ELSE
	tower_lamp.iol_slave_pdo_output.seg_1_color := 0; 
	tower_lamp.iol_slave_pdo_output.seg_2_color := 0; 
	tower_lamp.iol_slave_pdo_output.seg_3_color := 0; 
	
END_IF
*)
(*************************************************************************************
**************************************************************************************)

_handle_messages();
_write_output();

ACTION _handle_messages:
;
END_ACTION

ACTION _handle_process_test:
;
END_ACTION

ACTION _mode_manager:
IF process_mode_req_is_pending(CONVERSION_this := prc)
THEN
    process_apply_mode_req_first_step(CONVERSION_this := prc);
    CASE process_get_mode(CONVERSION_this := prc) OF
        MODE_TO_ABSENT:
            ;
        MODE_TO_INACTIVE:
            ;
        MODE_TO_TEST:
            ;
        MODE_TO_OPERATIONAL:
            ;
    END_CASE
    process_apply_mode_req_second_step(CONVERSION_this := prc);
END_IF;
END_ACTION

ACTION _objects_manager:
IF objects_initialization()
THEN
    sub_process_init(
        object_name 				:= 'csp_main_services_towerLamp.prc',
        process						:= csp_main_services.prc,
        CONVERSION_this				:= prc);

	prc_path 						:= process_get_path(prc);

	digital_output_init(
		object_name 				:= CONCAT(prc_path, '_buzzer_do'),
		polarity_direct				:= TRUE,
		process 					:= prc,
		CONVERSION_this 			:= buzzer_do);
		
	lamp_init(
		object_name 				:= CONCAT(prc_path, '_buzzer_lmp'),
		process 					:= prc,
		dout						:= buzzer_do,
		CONVERSION_this 			:= buzzer_lmp);
	
	filter_init(
		object_name := CONCAT(prc_path, '_buzzer_filt'),
		delay_off_on := 0,
		delay_on_off := 3000, //Marco: it's equal to the half of the desired buzzer timer (i.e. desired 1.5s --> delay = 3 s)
		process := prc,
		CONVERSION_this := buzzer_filt);
	
		(* BUZZER CONDITIONER *)
	motorization_conditioner_init(
		object_name					:= CONCAT(prc_path, '_buzzer_motcond'),
		velocity_limit				:= 0.0,
		velocity_limit_active		:= FALSE,
		idle_handshake_active		:= FALSE,
		execute_handshake_active	:= TRUE,
		hold_handshake_active		:= FALSE,
		suspend_handshake_active	:= FALSE,
		complete_handshake_active	:= FALSE,
		abort_handshake_active		:= FALSE,
		stop_handshake_active		:= FALSE,
		origin						:= MOTORIZATION_CONDITIONER_ORIGIN_INTERNAL,
		manager						:= csp_main_motorization_manager.motm,
		process						:= prc,
		CONVERSION_this				:= buzzer_motcond);

	boolean_or_init(
		object_name 				:= CONCAT(prc_path, '_buzzer_req_bool_or'),
		process 					:= prc,
		CONVERSION_this 			:= buzzer_req_bool_or);
	
	(* boolean_init(            
		object_name					:= CONCAT(prc_path, '_buzzer_status_bool'), 
		process						:= prc, 
		CONVERSION_this				:= buzzer_status_bool);
		
	signaling_device_configure_buzzer_behaviour(
		working_mode:= SIGNALING_DEVICE_BUZZER_WORKING_MODE_STATE_ON_OFF, 
		custom_pwm_period_ms:= 0, 
		buzzer_time_to_exec_from_starting:=3000 , 
		buzzer_time_to_exec_from_unholding:= 300, 
		CONVERSION_this:=tower_lamp );

	timer_init(
		object_name					:= CONCAT(prc_path, '_buzzer_tmr'),
		process						:= prc,
	    CONVERSION_this				:= buzzer_tmr);


		*)	
		
	signaling_device_iol_balluff_init(
		object_name 				:= CONCAT(prc_path, '_tower_lamp'),
		master_channel 				:= 1,
		blue_light_enable 			:= TRUE,
		white_light_enable 			:= TRUE,
		io_link_master 				:= csp_main_services.iol_master_el6224_IO6100,
		machine 					:= csp.mch,
		buzzer 						:= buzzer_lmp,
		process 					:= prc,
		CONVERSION_this 			:= tower_lamp);
	
	filter_init(
		object_name 				:= CONCAT(prc_path, '_reject_status_flt'),
		delay_off_on				:= flt_timer_off_on,
		delay_on_off 				:= flt_timer_on_off,
		process			 			:= prc,
		CONVERSION_this 			:= reject_status_flt);	
	
	parameter_overwrite_bool_init(
		object_name								:= CONCAT(prc_path, '_reject_ack_overwrite'),
		parameter								:= Reject_Acknowledged,
		process									:= prc,
		CONVERSION_this							:= reject_ack_overwrite);
	
	
END_IF;

IF	objects_running()
THEN
	process_cycle(prc);
	lamp_cycle(buzzer_lmp);
	
	filter_cycle(input:= buzzer_req_bool, buzzer_filt);
	filter_cycle(input:= reject_present_filtered,	CONVERSION_this := reject_status_flt);	
		
	signaling_device_cycle(tower_lamp);
	motorization_conditioner_cycle(buzzer_motcond);
END_IF;
END_ACTION

ACTION _read_process_image:
;
END_ACTION

ACTION _read_var_input:
;
END_ACTION

ACTION _set_runtime_properties:
;
END_ACTION

ACTION _sim_update:
;
END_ACTION

ACTION _write_output:
(* SIMULATION *)
;
END_ACTION

END_PROGRAM

// ---- Application/CSP/Main/Services/csp_main_services.TcPOU
(********************* G.D S.p.A. - Technical Department *****************************

Date			Version		Author			Description             
----------      -------		-----------		----------------------------------------------
2015/06/30		0000.00		M.Grasso		Initial Release

DESCRIPTION:	

NOTES:        		 

**************************************************************************************)
(*$R process_ref := prc; $*)

PROGRAM csp_main_services
VAR
	prc:								process;
	prc_path:							STRING;
	reset_output_test:					digital_output;
	
	iol_master_el6224_IO6100:			iol_master;
	
	lights_toggle:						BOOL := TRUE; (*$P $*)
	
	pressure_switch_value AT %I*:		INT;
	no_pressure_dchk:					digital_check;
	pressure_level_low_bool:			boolean;
	pressure_value_limit:				INT := 1000; (*$P $*)
	pressure_check_delay:				DINT := 15000; (*$P $*)
	
	air_not_above_limit_motcond:		motorization_conditioner;
	
	pressure_check_delay_running: 		DINT := 100;
END_VAR

_read_var_input();
_objects_manager();

IF g_application_status <> APPLICATION_STATUS_RUNNING
THEN
	RETURN;
END_IF

_read_process_image();

_mode_manager();

CASE process_get_mode (CONVERSION_this := prc) OF

	MODE_ABSENT,
	MODE_INACTIVE:
		RETURN;

	MODE_TEST:
		_handle_process_test();
END_CASE
_set_runtime_properties();

(*************************************************************************************
**************************************************************************************)
(*BODY*)

IF descriptor_get_reset_edge(prc.descriptor)
THEN
	digital_output_set(reset_output_test);
ELSE
	digital_output_reset(reset_output_test);
END_IF



(* LOGIC TO CHECK FOR PRESSURE AFTER MACHINE IS READY *)
IF machine_is_running(csp.mch)
AND pressure_switch_value < pressure_value_limit
	THEN
		digital_check_set_alarm_delay(
			alarm_delay := pressure_check_delay_running,
			CONVERSION_this := no_pressure_dchk);
		boolean_set(pressure_level_low_bool);
END_IF

IF machine_is_ready(csp.mch)
AND pressure_switch_value < pressure_value_limit
	THEN
digital_check_set_alarm_delay(
	alarm_delay := pressure_check_delay,
	CONVERSION_this := no_pressure_dchk);
		boolean_set(pressure_level_low_bool);
END_IF


IF machine_is_stopped(csp.mch)
	OR 
	pressure_switch_value > pressure_value_limit
	THEN
	boolean_reset(pressure_level_low_bool);
END_IF



IF	motorization_manager_is_starting(csp_main_motorization_manager.motm)
AND pressure_switch_value > pressure_value_limit
	THEN
		motorization_conditioner_start_done(air_not_above_limit_motcond);
END_IF

(*************************************************************************************
**************************************************************************************)

_handle_messages();
_write_output();

ACTION _handle_messages:
;
END_ACTION

ACTION _handle_process_test:
;
END_ACTION

ACTION _mode_manager:
IF process_mode_req_is_pending(CONVERSION_this := prc)
THEN
    process_apply_mode_req_first_step(CONVERSION_this := prc);
    CASE process_get_mode(CONVERSION_this := prc) OF
        MODE_TO_ABSENT:
            ;
        MODE_TO_INACTIVE:
            ;
        MODE_TO_TEST:
            ;
        MODE_TO_OPERATIONAL:
            ;
    END_CASE
    process_apply_mode_req_second_step(CONVERSION_this := prc);
END_IF;
END_ACTION

ACTION _objects_manager:
IF objects_initialization()
THEN
    sub_process_init(
	    object_name 	:= 'csp_main_services.prc',
        process			:= csp_main.prc,
        CONVERSION_this			:= prc);

	prc_path 			:= process_get_path(prc);

	digital_output_init(
		object_name		:= CONCAT(prc_path, '_reset_output_test'),
		polarity_direct	:= TRUE,
		process			:= prc,
		CONVERSION_this	:= reset_output_test);
		
	iol_master_init(
		object_name := 			'iol_master_el6224_IO6100',
		device_name := 			'SPLC5000Slot19 (EL6224)',
		_type := 				IOL_MASTER_BECKHOFF_EL6224,
		ethercat_master :=		csp_main.cabinet_ethercat_master,
		process := 				prc,
		CONVERSION_this := 		iol_master_el6224_IO6100);
		
		
	digital_check_and_message_init(
		object_name			:= CONCAT(prc_path, '_no_pressure_dchk'),
		alarm_if_input_off	:= FALSE,
		alarm_delay			:= pressure_check_delay,
		enabled_at_powerup	:= TRUE,
		individual_reset	:= FALSE,
		machine_reaction	:= MACHINE_REACTION_EMERGENCY_STOP,
		typology			:= MESSAGE_TYPOLOGY_EMERGENCY,
		process				:= prc,
		CONVERSION_this		:= no_pressure_dchk);

	boolean_init(
		object_name			:= CONCAT(prc_path, '_pressure_level_boolean'),
		process				:= prc,
		CONVERSION_this		:= pressure_level_low_bool);

	digital_check_add_boolean(
		boolean				:= pressure_level_low_bool,
		CONVERSION_this		:= no_pressure_dchk);

		
	motorization_conditioner_init(
		object_name					:=	CONCAT(prc_path, '_air_not_above_limit_motcond'),
		velocity_limit				:=	0.0,
		velocity_limit_active		:=	FALSE,
		idle_handshake_active		:=	FALSE,
		execute_handshake_active	:=	TRUE,
		hold_handshake_active		:=	FALSE,
		suspend_handshake_active	:=	FALSE,
		complete_handshake_active	:=	FALSE,
		abort_handshake_active		:=	FALSE,
		stop_handshake_active		:=	FALSE,
		origin						:=	MOTORIZATION_CONDITIONER_ORIGIN_INTERNAL,
		manager						:=	csp_main_motorization_manager.motm,
		process						:=	prc,
		CONVERSION_this				:=	air_not_above_limit_motcond);
		
END_IF

IF objects_running()
THEN
	process_cycle(prc);
	iol_master_cycle(iol_master_el6224_IO6100);
	digital_check_cycle(no_pressure_dchk);
	motorization_conditioner_cycle(air_not_above_limit_motcond);
END_IF
END_ACTION

ACTION _read_process_image:
;
END_ACTION

ACTION _read_var_input:
;
END_ACTION

ACTION _set_runtime_properties:
;
END_ACTION

ACTION _write_output:
;
END_ACTION

END_PROGRAM

// ---- Application/CSP/Case/Feed/Kinematic/csp_case_feed_kinematic_y.TcPOU
(*********************************** G.D S.p.A. - Technical Department ***********************************
============= PROGRAM INFO ============
FOLDER:             TBD
MACHINES INVOLVED:  TBD 

============= DESCRIPTION =============
csp machine declaration

============= REVISIONS ===============
Date		Version	 	Author      	Description             
----------	-------		------------  	--------------------------------------------
2019/04/05 	0000.00	 	M.Grasso		Creation of the PRG

**********************************************************************************************************)
(*$R process_ref := prc; $*)
PROGRAM csp_case_feed_kinematic_y
VAR
		
	prc:												process;
	prc_path:											STRING;
	
	axis:												axis;
	axis_actual_position:								LREAL;

	fsm_enable_condition:								BOOL := FALSE;
	fsm_next_status:									csp_case_feed_kinematic_status_enum;
	fsm_status:											csp_case_feed_kinematic_status_enum;
	debug_state_machine:								BOOL := FALSE;
	debug_state_machine_one_step:						BOOL := FALSE;	
	
	in_accu_safe_pos:                                   BOOL := FALSE;
    accu_tolerance:                                     LREAL := 5.0;
    accu_safe_pos:                                      LREAL := -485;
	
	cam_id:												INT := 3;
	
	local_test: BOOL := false;
END_VAR

VAR CONSTANT
	MOTOR_PHASE_VELOCITY_MMPS:							LREAL := 20;	
	MOTOR_MAX_VELOCITY_MMPS:							LREAL := 1000;
	MOTOR_MAX_ACCELLERATION_MMPS2:						LREAL := 10000;
	MOTOR_MAX_DECELLERATION_MMPS2:						LREAL := 10000;
	MOTOR_MAX_JERK_MMPS3:								LREAL := 100000; 
	MOTOR_MAX_FOLLOWING_ERROR_MM:						LREAL := 10;
END_VAR

_read_var_input();

_object_manager();

IF NOT objects_running()
THEN
	RETURN;	
END_IF

_read_process_image();

_mode_manager();

CASE process_get_mode(prc) OF
	MODE_ABSENT,
	MODE_INACTIVE:
		RETURN;
	MODE_TEST:
		_handle_process_test();
END_CASE

_set_runtime_properties();

(********************************* BODY *********************************)

IF (axis.actual_position > (accu_safe_pos - accu_tolerance)) AND axis.actual_position < (accu_safe_pos + accu_tolerance)
THEN
	in_accu_safe_pos := TRUE;
ELSE
	in_accu_safe_pos := FALSE;   
END_IF

// Manage the accu change safe position
fsm_enable_condition := axis_is_ok(FALSE, axis)	
						AND															
						(csp_case_feed_kinematic.fsm_status = CSP_CASE_FEED_KINEMATIC_STATUS_ENABLED)
						AND
						csp_case_feed_kinematic.cartesian_mode_active
						AND							
						csp_main_accuChange.Brand_Change_Occurred;
										
IF	NOT fsm_enable_condition
	AND
	fsm_status <> CSP_CASE_FEED_KINEMATIC_STATUS_DISABLED	
THEN
	fsm_next_status	:= CSP_CASE_FEED_KINEMATIC_STATUS_DISABLED;
END_IF
					
CASE fsm_status OF
	
	CSP_CASE_FEED_KINEMATIC_STATUS_NOT_INITIALIZED:
	
        IF	axis_is_ok(return_when_absent := TRUE, CONVERSION_this := axis)
        THEN
            fsm_next_status := CSP_CASE_FEED_KINEMATIC_STATUS_DISABLED;
        END_IF

		
	CSP_CASE_FEED_KINEMATIC_STATUS_DISABLED:
	
		IF	fsm_enable_condition
			AND
			motorization_conditioner_is_execute(csp_main_services_towerLamp.buzzer_motcond) 							
		THEN	
			IF	in_accu_safe_pos
			THEN
				fsm_next_status := CSP_CASE_FEED_KINEMATIC_STATUS_CHANGE_OVER_MODE_DONE;
			ELSE								
				fsm_next_status := CSP_CASE_FEED_KINEMATIC_STATUS_ENABLED;
			END_IF
		END_IF;

		
	CSP_CASE_FEED_KINEMATIC_STATUS_ENABLED:	
	
		axis_move_absolute(
			position 		:= accu_safe_pos,
			velocity 		:= MOTOR_PHASE_VELOCITY_MMPS,
			direction		:= AXIS_CURRENT_DIRECTION,
			acceleration 	:= MOTOR_MAX_ACCELLERATION_MMPS2,
			deceleration 	:= MOTOR_MAX_DECELLERATION_MMPS2,
			jerk 			:= MOTOR_MAX_JERK_MMPS3, 
			buffer_mode 	:= AXIS_BUFFER_MODE_BUFFERED,
			CONVERSION_this := axis);
			
		IF 	axis_is_absolute_moving(axis)
		THEN
			fsm_next_status	:= CSP_CASE_FEED_KINEMATIC_STATUS_CHANGE_OVER_MODE;
		END_IF
		
		
	CSP_CASE_FEED_KINEMATIC_STATUS_CHANGE_OVER_MODE:

		IF 	axis_is_standstill(axis)
		THEN	
			axis_disable(axis);					
			fsm_next_status := CSP_CASE_FEED_KINEMATIC_STATUS_CHANGE_OVER_MODE_DONE;
		END_IF
		
		
	CSP_CASE_FEED_KINEMATIC_STATUS_CHANGE_OVER_MODE_DONE:
		;
		
END_CASE

IF 	NOT debug_state_machine
	OR
	debug_state_machine_one_step
THEN
	fsm_status := fsm_next_status;
	debug_state_machine_one_step := FALSE;
END_IF

(* TEMPORARY CAM CHANGE *)
IF csp_main_brand.count = '24Count'
	THEN
		cam_id := 503; //beta 1,3,10 = 303; beta 4 = 503; alpha 1 = 403
ELSIF csp_main_brand.count = '10Count'
	THEN
		cam_id := 572;
ELSIF csp_main_brand.count = '32Count'
	THEN
		cam_id := 3;
ELSIF csp_main_brand.count = '48Count'
	THEN
		cam_id := 44;
END_IF

(************************************************************************)

_handle_messages();

_write_output();

ACTION _handle_messages:
;
END_ACTION

ACTION _handle_process_test:
;
END_ACTION

ACTION _mode_manager:
IF process_mode_req_is_pending(prc)
THEN
    process_apply_mode_req_first_step(prc);
    CASE process_get_mode(prc) OF
        MODE_TO_ABSENT:
			;
        MODE_TO_INACTIVE:
			;
        MODE_TO_TEST:
			;
        MODE_TO_OPERATIONAL:
			;
    END_CASE
    process_apply_mode_req_second_step(prc);
END_IF
END_ACTION

ACTION _object_manager:
IF objects_initialization()
THEN
	sub_process_init(
		object_name					:= 'csp_case_feed_kinematic_y.prc', 
		process						:= csp_case_feed_kinematic.prc, 
		CONVERSION_this				:= prc);
		
	prc_path 						:= process_get_path(prc);
	
	axis_init(
		object_name					:= CONCAT(prc_path, '_axis'), 
		axis_type					:= AXIS_TYPE_VIRTUAL, 
		encoder_scaling_factor		:= G_VIRTUAL_ENCODER_SCALING_FACTOR_DEGPINC,
		modulo						:= G_NO_MODULO_DEG, 
		process						:= prc, 
		CONVERSION_this				:= axis);
	
	axis_set_max_dynamic(
		reference_velocity			:=	MOTOR_MAX_VELOCITY_MMPS,
		velocity					:=	MOTOR_MAX_VELOCITY_MMPS,
		acceleration				:=	MOTOR_MAX_ACCELLERATION_MMPS2,
		deceleration				:=	MOTOR_MAX_DECELLERATION_MMPS2,
		jerk						:=	MOTOR_MAX_JERK_MMPS3,
		following_error				:=	MOTOR_MAX_FOLLOWING_ERROR_MM,
		CONVERSION_this				:=	axis);
		

END_IF

IF objects_running()
THEN
	process_cycle(prc);
	axis_cycle(axis);
END_IF
END_ACTION

ACTION _read_process_image:
;
END_ACTION

ACTION _read_var_input:
;
END_ACTION

ACTION _set_runtime_properties:
axis_actual_position := axis_get_actual_incremental_position(axis);
END_ACTION

ACTION _write_output:
;
END_ACTION

END_PROGRAM

// ---- Application/CSP/Case/Feed/Kinematic/csp_case_feed_kinematic_tilt.TcPOU
(*********************************** G.D S.p.A. - Technical Department ***********************************
============= PROGRAM INFO ============
FOLDER:             TBD
MACHINES INVOLVED:  TBD 

============= DESCRIPTION =============
csp machine declaration

============= REVISIONS ===============
Date		Version	 	Author      	Description             
----------	-------		------------  	--------------------------------------------
2019/04/05 	0000.00	 	M.Grasso		Creation of the PRG

**********************************************************************************************************)
(*$R process_ref := prc; $*)
PROGRAM csp_case_feed_kinematic_tilt
VAR
		
	prc:												process;
	prc_path:											STRING;
	
	axis:												axis;
	axis_actual_position:								LREAL;
	
	fsm_enable_condition:								BOOL := FALSE;
	fsm_next_status:									csp_case_feed_kinematic_status_enum;
	fsm_status:											csp_case_feed_kinematic_status_enum;
	debug_state_machine:								BOOL := FALSE;
	debug_state_machine_one_step:						BOOL := FALSE;	
	
	in_accu_safe_pos:                                   BOOL := FALSE;
    accu_tolerance:                                     LREAL := 5.0;
    accu_safe_pos:                                      LREAL := 1334.5;
	
	cam_id:												INT := 7;

	local_test: 										BOOL := false;
END_VAR

VAR CONSTANT
	MOTOR_PHASE_VELOCITY_DEGPS:							LREAL := 8;	
	MOTOR_MAX_VELOCITY_DEGPS:							LREAL := 9600;
	MOTOR_MAX_ACCELLERATION_DEGPS2:						LREAL := 4800;
	MOTOR_MAX_DECELLERATION_DEGPS2:						LREAL := 4800;
	MOTOR_MAX_JERK_DEGPS3:								LREAL := 100000000; 
	MOTOR_MAX_FOLLOWING_ERROR_DEG:						LREAL := 2;
END_VAR

_read_var_input();

_object_manager();

IF 	NOT objects_running()
THEN
	RETURN;	
END_IF

_read_process_image();

_mode_manager();

CASE process_get_mode(prc) OF
	MODE_ABSENT,
	MODE_INACTIVE:
		RETURN;
	MODE_TEST:
		_handle_process_test();
END_CASE

_set_runtime_properties();

(********************************* BODY *********************************)

IF (axis.actual_position > (accu_safe_pos - accu_tolerance)) AND axis.actual_position < (accu_safe_pos + accu_tolerance)
THEN
	in_accu_safe_pos := TRUE;
ELSE
	in_accu_safe_pos := FALSE;   
END_IF

// Manage the accu change safe position
fsm_enable_condition := axis_is_ok(FALSE, axis)	
						AND															
						(csp_case_feed_kinematic.fsm_status = CSP_CASE_FEED_KINEMATIC_STATUS_ENABLED)
						AND
						csp_case_feed_kinematic.cartesian_mode_active
						AND							
						csp_main_accuChange.Brand_Change_Occurred;
										
IF	NOT fsm_enable_condition
	AND
	fsm_status <> CSP_CASE_FEED_KINEMATIC_STATUS_DISABLED	
THEN
	fsm_next_status	:= CSP_CASE_FEED_KINEMATIC_STATUS_DISABLED;
END_IF
					
CASE fsm_status OF
	
	CSP_CASE_FEED_KINEMATIC_STATUS_NOT_INITIALIZED:
	
        IF	axis_is_ok(return_when_absent := TRUE, CONVERSION_this := axis)
        THEN
            fsm_next_status := CSP_CASE_FEED_KINEMATIC_STATUS_DISABLED;
        END_IF
		

	CSP_CASE_FEED_KINEMATIC_STATUS_DISABLED:
	
		IF	fsm_enable_condition
			AND
			motorization_conditioner_is_execute(csp_main_services_towerLamp.buzzer_motcond) 							
		THEN	
			IF	in_accu_safe_pos
			THEN
				fsm_next_status := CSP_CASE_FEED_KINEMATIC_STATUS_CHANGE_OVER_MODE_DONE;
			ELSE								
				fsm_next_status := CSP_CASE_FEED_KINEMATIC_STATUS_ENABLED;
			END_IF
		END_IF;
		

	CSP_CASE_FEED_KINEMATIC_STATUS_ENABLED:	
	
		axis_move_absolute(
			position 		:= accu_safe_pos,
			velocity 		:= MOTOR_PHASE_VELOCITY_DEGPS,
			direction		:= AXIS_CURRENT_DIRECTION,
			acceleration 	:= MOTOR_MAX_ACCELLERATION_DEGPS2,
			deceleration 	:= MOTOR_MAX_DECELLERATION_DEGPS2,
			jerk 			:= MOTOR_MAX_JERK_DEGPS3, 
			buffer_mode 	:= AXIS_BUFFER_MODE_BUFFERED,
			CONVERSION_this := axis);
			
		IF 	axis_is_absolute_moving(axis)
		THEN
			fsm_next_status	:= CSP_CASE_FEED_KINEMATIC_STATUS_CHANGE_OVER_MODE;
		END_IF
		
		
	CSP_CASE_FEED_KINEMATIC_STATUS_CHANGE_OVER_MODE:
	
		IF 	axis_is_standstill(axis)
		THEN	
			axis_disable(axis);					
			fsm_next_status := CSP_CASE_FEED_KINEMATIC_STATUS_CHANGE_OVER_MODE_DONE;
		END_IF
		
	CSP_CASE_FEED_KINEMATIC_STATUS_CHANGE_OVER_MODE_DONE:
	
		;
		
END_CASE

IF 	NOT debug_state_machine
	OR
	debug_state_machine_one_step
THEN
	fsm_status := fsm_next_status;
	debug_state_machine_one_step := FALSE;
END_IF


(* TEMPORARY CAM CHANGE *)
IF csp_main_brand.count = '24Count'
	THEN
		cam_id := 307;
ELSIF csp_main_brand.count = '10Count'
	THEN
		cam_id := 573;
ELSIF csp_main_brand.count = '32Count'
	THEN
		cam_id := 7;
ELSIF csp_main_brand.count = '48Count'
	THEN
		cam_id := 45;
END_IF

(************************************************************************)

_handle_messages();

_write_output();

ACTION _handle_messages:
;
END_ACTION

ACTION _handle_process_test:
;
END_ACTION

ACTION _mode_manager:
IF process_mode_req_is_pending(prc)
THEN
    process_apply_mode_req_first_step(prc);
    CASE process_get_mode(prc) OF
        MODE_TO_ABSENT:
			;
        MODE_TO_INACTIVE:
			;
        MODE_TO_TEST:
			;
        MODE_TO_OPERATIONAL:
			;
    END_CASE
    process_apply_mode_req_second_step(prc);
END_IF
END_ACTION

ACTION _object_manager:
IF objects_initialization()
THEN
	sub_process_init(
		object_name					:= 'csp_case_feed_kinematic_tilt.prc', 
		process						:= csp_case_feed_kinematic.prc, 
		CONVERSION_this				:= prc);
		
	prc_path 						:= process_get_path(prc);
	
	axis_init(
		object_name					:= CONCAT(prc_path, '_axis'), 
		axis_type					:= AXIS_TYPE_VIRTUAL, 
		encoder_scaling_factor		:= G_VIRTUAL_ENCODER_SCALING_FACTOR_DEGPINC,
		modulo						:= G_NO_MODULO_DEG, 
		process						:= prc, 
		CONVERSION_this				:= axis);
	
	axis_set_max_dynamic(
		reference_velocity			:=	MOTOR_MAX_VELOCITY_DEGPS,
		velocity					:=	MOTOR_MAX_VELOCITY_DEGPS,
		acceleration				:=	MOTOR_MAX_ACCELLERATION_DEGPS2,
		deceleration				:=	MOTOR_MAX_DECELLERATION_DEGPS2,
		jerk						:=	MOTOR_MAX_JERK_DEGPS3,
		following_error				:=	MOTOR_MAX_FOLLOWING_ERROR_DEG,
		CONVERSION_this				:=	axis);
	

END_IF

IF objects_running()
THEN
	process_cycle(prc);
	axis_cycle(axis);
END_IF
END_ACTION

ACTION _read_process_image:
;
END_ACTION

ACTION _read_var_input:
;
END_ACTION

ACTION _set_runtime_properties:
axis_actual_position := axis_get_actual_incremental_position(axis);
END_ACTION

ACTION _write_output:
;
END_ACTION

END_PROGRAM

// ---- POUs/AFL extensions/jog_manager/commands/jog_manager_reset_pendant_active.TcPOU
(*$
	Reset the pendant activation to ogject <b><i>this</i></b>.
	The method returns <i>TRUE</i> if the command is accepted, otherwise it returns <i>FALSE</i>.
$*)
FUNCTION jog_manager_reset_pendant_active : BOOL
VAR_INPUT	
END_VAR
VAR_IN_OUT
    CONVERSION_this:		jog_manager;	(*$ Instance to which the method applies $*)
END_VAR

IF	NOT (descriptor_mode_is_operational(CONVERSION_this.descriptor)
		(*OR
		descriptor_mode_is_test(CONVERSION_this.descriptor)*))
THEN
	jog_manager_reset_pendant_active := FALSE;				(* command rejected *)
 	RETURN;
END_IF

parameter_overwrite_set_bool_value(FALSE, CONVERSION_this.pendant_active_pow);

jog_manager_reset_pendant_active := TRUE;					(* command accepted *)

END_FUNCTION

// ---- POUs/AFL extensions/jog_manager/status/jog_manager_is_pendant_active.TcPOU
(*$
	Returns <i>pendant_active</i> of the instance <b><i>this</i></b>.
	Returns always false if pendant is not present.
$*)
FUNCTION jog_manager_is_pendant_active: BOOL
VAR_IN_OUT
    CONVERSION_this:	jog_manager;	(*$ Instance to which the method applies $*)
END_VAR

jog_manager_is_pendant_active := 
	CONVERSION_this.has_pendant
	AND
	CONVERSION_this.pendant_active;

END_FUNCTION

// ---- Application/CSP/Case/Feed/csp_case_feed.TcPOU
(*********************************** G.D S.p.A. - Technical Department ***********************************
============= PROGRAM INFO ============
FOLDER:             TBD
MACHINES INVOLVED:  TBD 

============= DESCRIPTION =============
csp machine declaration

============= REVISIONS ===============
Date		Version	 	Author      	Description             
----------	-------		------------  	--------------------------------------------
2019/04/05 	0000.00	 	M.Grasso		Creation of the PRG

**********************************************************************************************************)
(*$R process_ref := prc; $*)
PROGRAM csp_case_feed
VAR
	
	prc:											process;
	prc_path:										STRING;
	
	Feed_request:									BOOL;
	case_at_loading_sr: 							DINT := 26;
END_VAR

_read_var_input();

_object_manager();

IF NOT objects_running()
THEN
	RETURN;	
END_IF

_read_process_image();

_mode_manager();

_set_runtime_properties();

(********************************* BODY *********************************)
IF (shift_register_step_has_status_item(
	step_id := case_at_loading_sr,
	status_bits_to_be_true := ITEM_HAS_LS_LOWER_FLAP + ITEM_HAS_LS_UPPER_FLAP + ITEM_HAS_OS_LOWER_FLAP + ITEM_HAS_OS_UPPER_FLAP,
	status_bits_to_be_false := 0,
	CONVERSION_this :=csp_case_main_statistics.sr)
   
	AND
	(csp_case_feed_virtualMaster.axis.actual_modulo_position > 340 
	AND NOT csp_case_loader_virtualMaster.product_loaded))   
	AND csp_case_loader.load_ready_at_loader	           
	THEN		 
		Feed_request :=FALSE;
	ELSIF NOT csp_case_transport_virtualMaster.stop_for_reject 
		THEN  
		Feed_request :=TRUE;
              
END_IF
(************************************************************************)

_handle_messages();

_write_output();

ACTION _handle_messages:
;
END_ACTION

ACTION _handle_process_test:
;
END_ACTION

ACTION _mode_manager:
IF process_mode_req_is_pending(prc)
THEN
    process_apply_mode_req_first_step(prc);
    CASE process_get_mode(prc) OF
        MODE_TO_ABSENT:
			;
        MODE_TO_INACTIVE:
			;
        MODE_TO_TEST:
			;
        MODE_TO_OPERATIONAL:
			;
    END_CASE
    process_apply_mode_req_second_step(prc);
END_IF
END_ACTION

ACTION _object_manager:
IF objects_initialization()
THEN
	sub_process_init(
		object_name					:= 'csp_case_feed.prc', 
		process						:= csp_case.prc, 
		CONVERSION_this				:= prc);
		
	prc_path 						:= process_get_path(prc);
END_IF

IF objects_running()
THEN
	process_cycle(prc);
END_IF
END_ACTION

ACTION _read_process_image:
;
END_ACTION

ACTION _read_var_input:
;
END_ACTION

ACTION _set_runtime_properties:
;
END_ACTION

ACTION _write_output:
;
END_ACTION

END_PROGRAM

// ---- Application/CSP/Case/csp_case.TcPOU
(*********************************** G.D S.p.A. - Technical Department ***********************************
============= PROGRAM INFO ============
FOLDER:             TBD
MACHINES INVOLVED:  TBD 

============= DESCRIPTION =============
csp machine declaration

============= REVISIONS ===============
Date		Version	 	Author      	Description             
----------	-------		------------  	--------------------------------------------
2019/04/05 	0000.00	 	M.Grasso		Creation of the PRG

**********************************************************************************************************)
(*$R process_ref := prc; $*)
PROGRAM csp_case
VAR
	
	prc:											process;
	prc_path:										STRING;
	disable_req:									BOOL:= FALSE;
	case_cammed_motcond:							motorization_conditioner;
	
	transport_engaged: 								BOOL;
	casefeed_engaged: 								BOOL;
END_VAR

_read_var_input();

_object_manager();

IF NOT objects_running()
THEN
	RETURN;	
END_IF

_read_process_image();

_mode_manager();

_set_runtime_properties();

(********************************* BODY *********************************)

disable_req := 	NOT machine_is_running(csp.mch)
				AND machine_is_stop_emergency_active(csp.mch)
				AND csp_main_motorization_virtualManager.axis.actual_velocity = 0;

				
(* Verifies tranfer virtual is cam engaged and allows motorization to start *)

IF //axis_is_cam_engaged(csp_case_virtualMaster.axis)
    csp_case_feed_virtualMaster.connection_done
	AND axis_is_cam_engaged(csp_case_feed_virtualMaster.axis)
    AND csp_case_transport_virtualMaster.transport_slaves_cammed
	AND csp_case_loader_virtualMaster.loader_slaves_cammed 
THEN
	motorization_conditioner_start_done(case_cammed_motcond);
END_IF
 

(* Axes engaged for jog management *) 
jog_manager_set_all_slave_axis_engaged(
	index					:= JOG_LIST_CSP_CASE_VIRTUAL, 
	all_slave_axis_engaged	:= 	axis_is_cam_engaged(csp_case_TRANSPORT_VIRTUALmASTER.axis)
							AND axis_is_cam_engaged(csp_case_FEED_VIRTUALMASTER.axis),
							//AND axis_is_cam_engaged(csp_case_LOADER_VIRTUALMASTER.axis),						 	
	CONVERSION_this			:= csp_main_jogManager.jog_manager_virtual);

	
	
IF axis_is_cam_engaged(csp_case_TRANSPORT_VIRTUALmASTER.axis)
THEN
	transport_engaged := TRUE;
ELSE
	transport_engaged := FALSE;	
END_IF

IF axis_is_cam_engaged(csp_case_FEED_VIRTUALMASTER.axis)
THEN
	casefeed_engaged := TRUE;
ELSE
	casefeed_engaged := FALSE;	
END_IF

	
(************************************************************************)

_handle_messages();

_write_output();

ACTION _handle_messages:
;
END_ACTION

ACTION _handle_process_test:
;
END_ACTION

ACTION _mode_manager:
IF process_mode_req_is_pending(prc)
THEN
    process_apply_mode_req_first_step(prc);
    CASE process_get_mode(prc) OF
        MODE_TO_ABSENT:
			;
        MODE_TO_INACTIVE:
			;
        MODE_TO_TEST:
			;
        MODE_TO_OPERATIONAL:
			;
    END_CASE
    process_apply_mode_req_second_step(prc);
END_IF
END_ACTION

ACTION _object_manager:
IF objects_initialization()
THEN
	process_init(
		object_name								:= 'csp_case.prc', 
		machine									:= csp.mch, 
		CONVERSION_this							:= prc);
		
	prc_path 									:= process_get_path(prc);
	
motorization_conditioner_init(
		object_name								:=	CONCAT(prc_path, '_case_cammed_motcond'),
		velocity_limit							:=	100.0,
		velocity_limit_active					:=	FALSE,
		idle_handshake_active					:=	FALSE,
		execute_handshake_active				:=	TRUE,
		hold_handshake_active					:=	FALSE,
		suspend_handshake_active				:=	FALSE,
		complete_handshake_active				:=	FALSE,
		abort_handshake_active					:=	FALSE,
		stop_handshake_active					:=	FALSE,
		origin									:=	MOTORIZATION_CONDITIONER_ORIGIN_INTERNAL,
		manager									:=	csp_main_motorization_manager.motm,
		process									:=	prc,
		CONVERSION_this							:=	case_cammed_motcond);
	
END_IF

IF objects_running()
THEN
	process_cycle(prc);
	motorization_conditioner_cycle(case_cammed_motcond);
END_IF
END_ACTION

ACTION _read_process_image:
;
END_ACTION

ACTION _read_var_input:
;
END_ACTION

ACTION _set_runtime_properties:
;
END_ACTION

ACTION _write_output:
;
END_ACTION

END_PROGRAM

// ---- POUs/AFL extensions/jog_manager/initialize/jog_manager_add_axis.TcPOU
(*$
	Adds the <a href="#axis_object"><i>axis_input</i></a> that performs 
	the jog command to the instance specified by the parameter <i><b>this</i></b>.
	<p>
	This function should be called at startup only.<br/>	
	Against errors on the input parameters the cpu is stopped, in this case the cause <br/>
	can be inspected in the global struct <i>framework.abort_error</i>: <br/>
	<br/>
    <li> <b>ERRORID_1 = 2</b>: <b><i>this</i></b> index outside boud </li>
    <li> <b>ERRORID_1 = 3</b>: <b><i>this</i></b> instance, index already defined </li>
	</p>
$*)
FUNCTION jog_manager_add_axis: VOID
VAR_INPUT
	list_index:			UINT;
						(*$ list index inside the jog_manager structure $*)
	master_axis:		BOOL;
						(*$ axis is master axis of some slaves $*)
	jog_type:			jog_manager_type;
						(*$ jog type allowed $*)
	sw_limit_positive:	LREAL;
						(*$ positive sw limit $*)
	sw_limit_negative:	LREAL;
						(*$ negative sw limit $*)
END_VAR
VAR_IN_OUT		
	axis:				axis;				(*$ <a href="#axis_object"><i>axis</i></a> membership $*)	
	CONVERSION_this:	jog_manager;		(*$ Instance to which the method applies $*)
END_VAR

IF 	(list_index <= JOG_MANAGER_JOG_LIST_NONE)
	OR
	(list_index > JOG_MANAGER_JOG_LIST_MAX)
THEN
 	abort(
		object_name := CONVERSION_this.object_name,
        errorID_1 := 2,
        errorID_2 := 0,
        errorID_3 := 0,
        error_str_1 := CONCAT(CONVERSION_this.object_name, ' list_index outside jog_manager boud'),
		error_str_2 := 'jog_manager_add_axis'
        );
    RETURN;
END_IF

IF 	CONVERSION_this.axis_list[list_index].axis = ADR(axis)
THEN
	RETURN;
END_IF

IF 	jog_manager_is_not_initialized(CONVERSION_this)
   	OR
   	axis_is_not_initialized(axis)
THEN
	IF 	framework_initialization()
	THEN
		RETURN;
	END_IF
END_IF

IF 	jog_manager_is_not_initialized(CONVERSION_this)
THEN
	framework_object_not_initialized_get_name(
		object_address := ADR(CONVERSION_this), 
		object_size := SIZEOF(CONVERSION_this),
		abort := TRUE,
		error_str_1 := 'object not initialized', 
		error_str_2 := 'jog_manager_add_axis'
	);
    RETURN;
END_IF

IF 	axis_is_not_initialized(axis)
THEN
	framework_object_not_initialized_get_name(
		object_address := ADR(axis), 
		object_size := SIZEOF(axis),
		abort := TRUE, 
		error_str_1 := 'object not initialized', 
		error_str_2 := CONCAT('Please check jog_manager_add_axis of ',CONVERSION_this.object_name)				
	);
    RETURN;
END_IF

IF 	(CONVERSION_this.axis_list[list_index].axis <> G_framework.NULL)
	AND
	(CONVERSION_this.axis_list[list_index].axis <> ADR(axis))
THEN
    abort(
		object_name := CONVERSION_this.object_name,
        errorID_1 := 3,
        errorID_2 := list_index,
        errorID_3 := 0,
        error_str_1 := CONCAT(CONVERSION_this.object_name, ' jog_manager has already axis in list'),
		error_str_2 := 'jog_manager_add_axis'
        );
    RETURN;
END_IF

CONVERSION_this.axis_list[list_index].axis := ADR(axis);
CONVERSION_this.axis_list[list_index].master_axis := master_axis;
CONVERSION_this.axis_list[list_index].jog_type := jog_type;
CONVERSION_this.axis_list[list_index].sw_limit_positive := sw_limit_positive;
CONVERSION_this.axis_list[list_index].sw_limit_negative := sw_limit_negative;

END_FUNCTION

// ---- Application/CSP/Case/Transport/csp_case_transport.TcPOU
(*********************************** G.D S.p.A. - Technical Department ***********************************
============= PROGRAM INFO ============
FOLDER:             TBD
MACHINES INVOLVED:  TBD 

============= DESCRIPTION =============
csp machine declaration
============= REVISIONS ===============
Date		Version	 	Author      	Description             
----------	-------		------------  	--------------------------------------------
2019/04/05 	0000.00	 	M.Grasso		Creation of the PRG

**********************************************************************************************************)
(*$R process_ref := prc; $*)
PROGRAM csp_case_transport
VAR
	
	 prc:                                            process;
    prc_path:                                        STRING;
    flap_dectect_sr:                                 INT:=25;
    case_at_loading_sr:                              INT:=26;
    transport_request:                               BOOL;
    //recovery_cycle:                                bool:= false;
    product_loaded:                                  BOOL;
	
	
	test_10: 										BOOL := FALSE;
	Followers_Extended: 							BOOL := FALSE;
	Followers_Spreaders_At_Starting_position: 		BOOL := FALSE;
	flap_control_axes_standstill: 					BOOL := FALSE;
	Spreaders_Extended: 							BOOL := false;
END_VAR

_read_var_input();

_object_manager();

IF NOT objects_running()
THEN
	RETURN;	
END_IF

_read_process_image();

_mode_manager();

_set_runtime_properties();

(********************************* BODY *********************************)
IF (shift_register_step_has_status_item(
	step_id := case_at_loading_sr,
	status_bits_to_be_true := ITEM_HAS_LS_LOWER_FLAP + ITEM_HAS_LS_UPPER_FLAP + ITEM_HAS_OS_LOWER_FLAP + ITEM_HAS_OS_UPPER_FLAP,
	status_bits_to_be_false := 0,
	CONVERSION_this :=csp_case_main_statistics.sr)
	AND
	NOT test_10)
THEN            
	transport_request :=FALSE;
ELSIF NOT csp_case_transport_virtualMaster.stop_for_reject 
THEN  
	transport_request :=TRUE;       
END_IF

IF (NOT csp_case_loader_virtualMaster.product_loaded
	OR NOT csp_case_loader_virtualMaster.At_Reject_product_loaded)
THEN
	test_10 := TRUE; //no product is loaded
ELSE
		test_10 := FALSE; // product is loaded
END_IF

(* Axes engaged for jog management *)
jog_manager_set_all_slave_axis_engaged(
	index					:= JOG_LIST_CSP_CASE_TRANSPORT_VIRTUAL, 
	all_slave_axis_engaged	:= 	axis_is_cam_engaged(csp_case_transport_os_trailing.axis)
							AND axis_is_cam_engaged(csp_case_transport_os_leading.axis)
							AND axis_is_cam_engaged(csp_case_transport_ls_trailing.axis)
							AND axis_is_cam_engaged(csp_case_transport_ls_leading.axis)
							//AND axis_is_cam_engaged(csp_case_tr_squaring_ls_leading.axis)
							AND axis_is_cam_engaged(csp_case_tr_squaring_ls_trailing.axis)
							AND axis_is_cam_engaged(csp_case_tr_squaring_os_leading.axis)
							AND axis_is_cam_engaged(csp_case_tr_squaring_os_trailing.axis)
							AND axis_is_cam_engaged(csp_case_closing_os_horizontal.axis)
							AND axis_is_cam_engaged(csp_case_closing_os_upper.axis)
							AND axis_is_cam_engaged(csp_case_closing_os_lower.axis)
							AND axis_is_cam_engaged(csp_case_closing_ls_horizontal.axis)
							AND axis_is_cam_engaged(csp_case_closing_ls_upper.axis)
							AND axis_is_cam_engaged(csp_case_closing_ls_lower.axis),						 	
	CONVERSION_this			:= csp_main_jogManager.jog_manager_virtual);
	
IF 	csp_case_fc_os_upper_follower.At_extended_position
	AND csp_case_fc_os_lower_follower.At_extended_position
	AND csp_case_fc_ls_upper_follower.At_extended_position
	AND csp_case_fc_ls_lower_follower.At_extended_position
THEN
	Followers_Extended := TRUE;
ELSE
	Followers_Extended := FALSE;	
END_IF

IF 	csp_case_fc_os_upper_spreader.At_extended_position
	AND csp_case_fc_os_lower_spreader.At_extended_position
	AND csp_case_fc_ls_upper_spreader.At_extended_position
	AND csp_case_fc_ls_lower_spreader.At_extended_position
THEN
	Spreaders_Extended := TRUE;
ELSE
	Spreaders_Extended := FALSE;	
END_IF

IF 	csp_case_fc_os_upper_follower.At_home_position
	AND csp_case_fc_os_lower_follower.At_home_position
	AND csp_case_fc_ls_upper_follower.At_home_position
	AND csp_case_fc_ls_lower_follower.At_home_position
	AND csp_case_fc_os_upper_spreader.At_home_position
	AND csp_case_fc_os_lower_spreader.At_home_position
	AND csp_case_fc_ls_upper_spreader.At_home_position
	AND csp_case_fc_ls_lower_spreader.At_home_position
THEN
	Followers_Spreaders_At_Starting_position := TRUE;
ELSE
	Followers_Spreaders_At_Starting_position := FALSE;
END_IF

IF 
axis_is_standstill(csp_case_fc_os_upper_spreader.axis) AND axis_is_standstill(csp_case_fc_os_upper_follower.axis)
AND axis_is_standstill(csp_case_fc_os_lower_spreader.axis) AND axis_is_standstill(csp_case_fc_os_lower_follower.axis)
AND axis_is_standstill(csp_case_fc_ls_lower_spreader.axis) AND axis_is_standstill(csp_case_fc_ls_lower_follower.axis)	
AND axis_is_standstill(csp_case_fc_ls_upper_spreader.axis) AND axis_is_standstill(csp_case_fc_ls_upper_follower.axis)
THEN
	flap_control_axes_standstill := TRUE;
ELSE
	flap_control_axes_standstill := FALSE;
END_IF
	
(************************************************************************)

_handle_messages();

_write_output();

ACTION _handle_messages:
;
END_ACTION

ACTION _handle_process_test:
;
END_ACTION

ACTION _mode_manager:
IF process_mode_req_is_pending(prc)
THEN
    process_apply_mode_req_first_step(prc);
    CASE process_get_mode(prc) OF
        MODE_TO_ABSENT:
			;
        MODE_TO_INACTIVE:
			;
        MODE_TO_TEST:
			;
        MODE_TO_OPERATIONAL:
			;
    END_CASE
    process_apply_mode_req_second_step(prc);
END_IF
END_ACTION

ACTION _object_manager:
IF objects_initialization()
THEN
	sub_process_init(
		object_name					:= 'csp_case_transport.prc', 
		process						:= csp_case.prc, 
		CONVERSION_this				:= prc);
		
	prc_path 						:= process_get_path(prc);
END_IF

IF objects_running()
THEN
	process_cycle(prc);
END_IF
END_ACTION

ACTION _read_process_image:
;
END_ACTION

ACTION _read_var_input:
;
END_ACTION

ACTION _set_runtime_properties:
;
END_ACTION

ACTION _write_output:
;
END_ACTION

END_PROGRAM

// ---- POUs/AFL extensions/jog_manager/status/jog_manager_is_jog_axis_deactivating.TcPOU
(*$
	Returns <i>TRUE</i> if the status of the instance <b><i>this</i></b> is
	<a href="#jog_manager_status_enum"><i>JOG_MANAGER_STATUS_ACTIVE</i></a>
	and  <i>list_selected</i> is a valid index,
	<i>FALSE</i> otherwise.
$*)
FUNCTION jog_manager_is_jog_axis_deactivating : BOOL
VAR_INPUT
	index:				UINT;
END_VAR
VAR_IN_OUT
    CONVERSION_this:	jog_manager;	(*$ Instance to which the method applies $*)
END_VAR

IF	(
		(CONVERSION_this.CONVERSION_private.list_selected <> CONVERSION_this.CONVERSION_private.old_list_selected)
		OR
		(CONVERSION_this.status = JOG_MANAGER_STATUS_SEL_DISABLE_AXIS)		
	)
	AND
	(CONVERSION_this.CONVERSION_private.old_list_selected = index)
	AND	
	CONVERSION_this.CONVERSION_private.old_list_selected_axis_is_valid
THEN
	jog_manager_is_jog_axis_deactivating := (CONVERSION_this.status >= JOG_MANAGER_STATUS_ACTIVE);
ELSE
	jog_manager_is_jog_axis_deactivating := FALSE;
END_IF

END_FUNCTION

// ---- Application/CSP/Case/Flap Control/csp_case_flapControl.TcPOU
(*********************************** G.D S.p.A. - Technical Department ***********************************
============= PROGRAM INFO ============
FOLDER:             TBD
MACHINES INVOLVED:  TBD 

============= DESCRIPTION =============
csp machine declaration

============= REVISIONS ===============
Date		Version	 	Author      	Description             
----------	-------		------------  	--------------------------------------------
2019/04/05 	0000.00	 	M.Grasso		Creation of the PRG

**********************************************************************************************************)
(*$R process_ref := prc; $*)
PROGRAM csp_case_flapControl
VAR
	
	prc:											process;
	prc_path:										STRING;
	Flap_check_begin_phase:							LREAL:=352;(*$P $*)
	Flap_check_end_phase:							LREAL:=357;(*$P $*)
	master_offset_all_followers:					LREAL := 2.4; (*$P $*)
	master_offset_all_spreaders:					LREAL := 355; (*$P $*)
	followers_spreaders_cammed:						motorization_conditioner;
	check_request_rtrig:							R_TRIG;
	check_request:									BOOL;
	
	bad_count:										INT := 0;
	consecutive_reject_aem:							message;
	
	consecutive_blocked_phwin:						phase_window;
	flap_check_on: 									LREAL := 180; (*$P $*)
	flap_check_off: 								LREAL := 250; (*$P $*)
	
	spreaders_clear: 								BOOL := TRUE;
END_VAR

_read_var_input();

_object_manager();

IF NOT objects_running()
THEN
	RETURN;	
END_IF

_read_process_image();

_mode_manager();

_set_runtime_properties();

(********************************* BODY *********************************)

IF axis_is_cam_engaged(csp_case_fc_os_lower_follower.axis)
	AND axis_is_cam_engaged(csp_case_fc_os_upper_follower.axis)
	AND axis_is_cam_engaged(csp_case_fc_os_lower_spreader.axis)
	AND axis_is_cam_engaged(csp_case_fc_os_upper_spreader.axis)
	AND axis_is_cam_engaged(csp_case_fc_ls_lower_follower.axis)
	AND axis_is_cam_engaged(csp_case_fc_ls_upper_follower.axis)
	AND axis_is_cam_engaged(csp_case_fc_ls_lower_spreader.axis)
	AND axis_is_cam_engaged(csp_case_fc_ls_upper_spreader.axis)
THEN
	motorization_conditioner_start_done(followers_spreaders_cammed);
END_IF


(* USED TO TRACK CONSECUTIVE REJECTS NO MATTER WHICH PE FAILS *)
check_request_rtrig(CLK := csp_case_feed_virtualMaster.follower_check_request);
check_request := check_request_rtrig.Q;

IF 	phase_window_falling_edge(csp_case_transport_virtualMaster.major_flap_phwin)
	OR	
	(
		check_request
		AND csp_case_transport.flap_control_axes_standstill
		AND csp_case_transport.Followers_Extended
		AND csp_case_transport.Spreaders_Extended
	)
THEN
	IF 	NOT digital_input_is_active(csp_case_fc_ls_lower_sensors.flap_di)
		OR NOT digital_input_is_active(csp_case_fc_ls_upper_sensors.flap_di)
		OR NOT digital_input_is_active(csp_case_fc_os_lower_sensors.flap_di)
		OR NOT digital_input_is_active(csp_case_fc_os_upper_sensors.flap_di)
		AND NOT csp_case_main_services.dry_cycle_mode
		AND NOT csp_main_motorization.empty_command	
	THEN
		bad_count :=  bad_count + 1;
	END_IF
	
END_IF


IF 	csp_case_transport_virtualMaster.PE_check
	OR machine_is_stopped(csp.mch)
	OR machine_is_stop_emergency_active(csp.mch)
THEN
	bad_count := 0;
	process_message_reset(consecutive_reject_aem);
END_IF


IF 	bad_count >= 3
	AND NOT csp_case_main_services.dry_cycle_mode
	AND NOT csp_main_motorization.empty_command
THEN
	process_message_set(1, 1, 1, consecutive_reject_aem);
END_IF



(* PHASE TO CHECK IF CONSECTUIVE BLOCKED PE *)
phase_window_set_phases_data(
	begin_phase:=  flap_check_on,
	end_phase:=  flap_check_off,
	begin_delay:= 0,
	end_delay:= 0,
	begin_max_compensation:= 0,
	end_max_compensation:= 0,
	CONVERSION_this:= consecutive_blocked_phwin);

IF 	csp_case_fc_ls_lower_spreader.in_accu_safe_pos 
	AND
	csp_case_fc_os_lower_spreader.in_accu_safe_pos
THEN 
	spreaders_clear := TRUE;
ELSE
	spreaders_clear := FALSE;
END_IF




(************************************************************************)

_handle_messages();

_write_output();

ACTION _handle_messages:
;
END_ACTION

ACTION _handle_process_test:
;
END_ACTION

ACTION _mode_manager:
IF process_mode_req_is_pending(prc)
THEN
    process_apply_mode_req_first_step(prc);
    CASE process_get_mode(prc) OF
        MODE_TO_ABSENT:
			;
        MODE_TO_INACTIVE:
			;
        MODE_TO_TEST:
			;
        MODE_TO_OPERATIONAL:
			;
    END_CASE
    process_apply_mode_req_second_step(prc);
END_IF
END_ACTION

ACTION _object_manager:
IF objects_initialization()
THEN
	sub_process_init(
		object_name					:= 'csp_case_flapControl.prc', 
		process						:= csp_case.prc, 
		CONVERSION_this				:= prc);
		
	prc_path 						:= process_get_path(prc);
	
	motorization_conditioner_init(
		object_name					:= CONCAT(prc_path, '_followers_spreaders_cammed'),
		velocity_limit				:= 0.0,
		velocity_limit_active		:= FALSE,
		idle_handshake_active		:= FALSE,
		execute_handshake_active	:= TRUE,
		hold_handshake_active		:= FALSE,
		suspend_handshake_active	:= FALSE,
		complete_handshake_active	:= FALSE,
		abort_handshake_active		:= FALSE,
		stop_handshake_active		:= FALSE,
		origin						:= MOTORIZATION_CONDITIONER_ORIGIN_INTERNAL,
		manager						:= csp_main_motorization_manager.motm,
		process						:= prc,
		CONVERSION_this				:= followers_spreaders_cammed);
	
	process_message_init(
		object_name:= CONCAT(prc_path, '_consecutive_reject_aem'), 
		behaviour:= MESSAGE_BEHAVIOUR_STATE, 
		reset_timeout:= 0, 
		disableable:= FALSE, 
		individual_reset:= FALSE, 
		machine_reaction:= MACHINE_REACTION_STOP_IN_PHASE_ONE, 
		typology:= MESSAGE_TYPOLOGY_ABNORMAL, 
		process:= prc, 
		CONVERSION_this:= consecutive_reject_aem);
		
		
	phase_window_init(
		object_name								:=CONCAT(PRC_PATH, '_consecutive_blocked_phwin'), 
		begin_phase								:=flap_check_on, 
		end_phase								:=flap_check_off, 
		begin_delay								:=0, 
		end_delay								:=0, 
		begin_max_compensation					:=0, 
		end_max_compensation					:=0, 
		generator								:=csp_case_transport_virtualMaster.transport_vm_phgen , 
		process									:=prc , 
		CONVERSION_this							:=consecutive_blocked_phwin);
		
END_IF

IF objects_running()
THEN
	process_cycle(prc);
	motorization_conditioner_cycle(followers_spreaders_cammed);
	phase_window_cycle(consecutive_blocked_phwin);
END_IF
END_ACTION

ACTION _read_process_image:
;
END_ACTION

ACTION _read_var_input:
;
END_ACTION

ACTION _set_runtime_properties:
;
END_ACTION

ACTION _write_output:
;
END_ACTION

END_PROGRAM

// ---- Application/CSP/Transfer/Crosspusher/csp_transfer_crosspusher.TcPOU
(*********************************** G.D S.p.A. - Technical Department ***********************************
============= PROGRAM INFO ============
FOLDER:             TBD
MACHINES INVOLVED:  TBD 

============= DESCRIPTION =============
csp machine declaration

============= REVISIONS ===============
Date		Version	 	Author      	Description             
----------	-------		------------  	--------------------------------------------
2019/04/05 	0000.00	 	M.Grasso		Creation of the PRG

**********************************************************************************************************)
(*$R process_ref := prc; $*)
PROGRAM csp_transfer_crosspusher
VAR
	
	prc:											process;
	prc_path:										STRING;
	
	loader_tolerance:								LREAL := 5; (*$P $*)
	loader_clear:									BOOL;
	loader_clear_test:								BOOL := FALSE;
	loader_home_position:							LREAL := 0;  (*$P $*) // MAYBE PULL VALUE FROM CSP_CASE_LOADER
	loader_status:									csp_transfer_crosspusher_loader_clear_status;
	
	debug_state_machine:							BOOL := FALSE;
	debug_reject_machine_one_step:					BOOL := FALSE;
	reject_status:									csp_transfer_crosspusher_reject_status_enum := CSP_TRANSFER_CROSSPUSHER_REJECT_STATUS_WAITING;
	reject_status_next:								csp_transfer_crosspusher_reject_status_enum := CSP_TRANSFER_CROSSPUSHER_REJECT_STATUS_WAITING;
	reject_done: 									BOOL;
	reject_running: 								BOOL;
	reject_dwell_transfer:							BOOL;
	reject_run_transfer:							BOOL;
	reject_time_out_tmr:							timer;	
	reject_status_last_state:						csp_transfer_crosspusher_reject_status_enum;
	e_stop_during_reject:							BOOL;
	
	
	horiz_to_follower_diff:							LREAL := 48; (*$P $*)
	horiz_to_follower_tolerance:					LREAL := 10; (*$P $*) // 15 for 10 count. 10 for 24 count
	
	calc_distance_between_pushers:					LREAL;
	distance_limit:									LREAL;
	distance_limit_tolerance:						LREAL := 50;
	follower_distance_to_horizontal_zero:			LREAL;
	pushers_too_close:								boolean;
	pushers_too_close_dchk:							digital_check;
	
	follower_pos_if_horiz_is_neg:					LREAL;
	follower_calc_pos:								LREAL;
	
	crosspusher_horiz_at_reject_low_limit:			LREAL;
	crosspusher_horiz_at_reject_high_limit:			LREAL;
	horizontal_reject_position:						LREAL := -400; (*$P $*)
	
	crosspusher_foll_at_reject_low_limit:			LREAL;
	crosspusher_foll_at_reject_high_limit:			LREAL;
	follower_reject_position:						LREAL := 845; (*$P $*)
	
	reject_velocity:								LREAL := 200; (*$P $*)
	
	cam_info_transfer:								axis_cam_info_data;
	cam_info_upstacker:								axis_cam_info_data;
	
	consecutive_accumulator_reject_asm:				message;
	temp1: 											BOOL;
	estop_occured_in_crosspush_reject: 				BOOL := False;
	calc_adjustment_for_follower: 					LREAL;
	
END_VAR
VAR_INPUT
	accumulator_reject_carton_count: 				DINT;(*$M $*)
	accumulator_reject_count: 						DINT;
END_VAR

_read_var_input();


_object_manager();

IF NOT objects_running()
THEN
	RETURN;	
END_IF

_read_process_image();

_mode_manager();

CASE process_get_mode(prc) OF
	MODE_ABSENT,
	MODE_INACTIVE:
		RETURN;
	MODE_TEST:
		_handle_process_test();
END_CASE
_set_runtime_properties();

(********************************* BODY *********************************)

(* STARTS REJECT SEQUENCE *)
crosspusher_horiz_at_reject_low_limit := horizontal_reject_position - 2;
crosspusher_horiz_at_reject_high_limit := horizontal_reject_position + 2;

crosspusher_foll_at_reject_low_limit := follower_reject_position - 2;
crosspusher_foll_at_reject_high_limit := follower_reject_position + 2;

IF csp_transfer_crosspusher_sensors.reject_stack
	AND NOT csp_transfer_upstacker_sensors.debug_active
THEN
	IF NOT reject_running
		THEN
		  reject_status_next := CSP_TRANSFER_CROSSPUSHER_REJECT_STATUS_START;
	END_IF		
END_IF

(* REJECT POU *)
reject();

IF reject_running
	AND NOT temp1
THEN
	temp1 := TRUE;
	accumulator_reject_carton_count := accumulator_reject_carton_count + 4;
	accumulator_reject_count := accumulator_reject_count +1;  // Added for consecutive crosspusher rejects
END_IF

//If the reject is not running the accumulator reject count is set to zero
IF (NOT reject_running
	AND csp_case_loader.load_ready_at_loader)
	OR csp_main_motorization.empty_command
THEN
	accumulator_reject_count := 0;
END_IF

//If accumulator is greater than 3 it will set the machine with an error
IF accumulator_reject_count >= 3
	AND NOT csp_main_motorization.empty_command
THEN
	process_message_set(0,0,0,consecutive_accumulator_reject_asm);
END_IF

// Clears consecutive accumulator rejects count and alarms once the machine is stopped.
IF (machine_is_stop_emergency_active(csp.mch)
	OR machine_is_stopped(csp.mch))
	AND process_message_is_on(consecutive_accumulator_reject_asm)
THEN
	process_message_reset(consecutive_accumulator_reject_asm);
	accumulator_reject_count := 0;
END_IF

IF NOT reject_running
THEN
	temp1 := FALSE;
END_IF	

(* JOG MANAGEMENT FO SLAVES *)
jog_manager_set_all_slave_axis_engaged(
	index					:= JOG_LIST_TRANSFER_CROSSPUSHER_VIRTUAL, 
	all_slave_axis_engaged	:= 	axis_is_cam_engaged(csp_transfer_crosspusher_horizontal.axis)
							   	AND
							   	axis_is_cam_engaged(csp_transfer_crosspusher_vertical.axis)
							 	AND
							 	axis_is_cam_engaged(csp_transfer_crosspusher_follower.axis),							 	
	CONVERSION_this			:= csp_main_jogManager.jog_manager_virtual);
 

(* VERIFIES LOADER IS CLEAR AND WILL NOT RUN *)
IF loader_clear_test
	OR ABS(csp_case_loader_pusher.axis.actual_position - loader_home_position) < loader_tolerance (* Loader is behind transfer section *)
THEN
	loader_clear := TRUE;
ELSE
	loader_clear := FALSE;
END_IF

(* SETS STATUS OF LOADER CLEAR ON PHASE EDGE *)
IF phase_edge(csp_transfer_crosspusher_virtualMaster.loader_clear_check_ph)
THEN
	loader_status := SEL(loader_clear, csp_transfer_crosspusher_loader_clear_status.NOT_CLEAR, csp_transfer_crosspusher_loader_clear_status.CLEAR);
ELSE
	loader_status := csp_transfer_crosspusher_loader_clear_status.NONE;
END_IF

(* USED FOR REJECT AND DISTANCE BETWEEN PADDLES *)
(* DISTANCE LIMIT CALCULATED BY THE CASE PATTERN AND CARTON DIMENSION MINUS THE TOLERANCE *)
distance_limit := csp_main_brand.carton_dimension.carton_size_L_mm * csp_main_brand.case_pattern.case_pattern_L - distance_limit_tolerance;
follower_distance_to_horizontal_zero := axis_get_actual_incremental_position(csp_transfer_crosspusher_follower.axis) - horiz_to_follower_diff;
calc_distance_between_pushers := follower_distance_to_horizontal_zero + axis_get_actual_incremental_position(csp_transfer_crosspusher_horizontal.axis);
calc_adjustment_for_follower := calc_distance_between_pushers - (csp_main_brand.carton_dimension.carton_size_L_mm * csp_main_brand.case_pattern.case_pattern_L + 40); //add 40mm for safety factor to keep distance ok		
follower_pos_if_horiz_is_neg := ABS(axis_get_actual_incremental_position(csp_transfer_crosspusher_horizontal.axis)) + horiz_to_follower_diff	+ csp_transfer_crosspusher_follower.slave_scaling;
		
(* STOPS MACHINE IF PUSHERS COME TOO CLOSE - USES AUTO CALCULATION DIFFERENCE *)
IF axis_is_moving(csp_main_motorization_virtualManager.axis)
	AND csp_transfer_crosspusher_follower.connection_done
	AND csp_transfer_crosspusher_horizontal.connection_done
	AND calc_distance_between_pushers < distance_limit
THEN
	boolean_set(pushers_too_close);
END_IF

(* CLEARS PUSHERS TOO CLOSE DIGITAL CHECK *)
IF NOT axis_is_moving(csp_main_motorization_virtualManager.axis)
THEN
	boolean_reset(pushers_too_close);
END_IF

(************************************************************************)

_handle_messages();

_write_output();

ACTION _handle_messages:
;
END_ACTION

ACTION _handle_process_test:
;
END_ACTION

ACTION _mode_manager:
IF process_mode_req_is_pending(prc)
THEN
    process_apply_mode_req_first_step(prc);
    CASE process_get_mode(prc) OF
        MODE_TO_ABSENT:
			;
        MODE_TO_INACTIVE:
			;
        MODE_TO_TEST:
			;
        MODE_TO_OPERATIONAL:
			;
    END_CASE
    process_apply_mode_req_second_step(prc);
END_IF
END_ACTION

ACTION _object_manager:
IF objects_initialization()
THEN
	sub_process_init(
		object_name					:= 'csp_transfer_crosspusher.prc', 
		process						:= csp_transfer.prc, 
		CONVERSION_this				:= prc);
		
	prc_path 						:= process_get_path(prc);
	
	
	boolean_init(
		object_name:= CONCAT(prc_path, '_pushers_too_close'), 
		process:= prc, 
		CONVERSION_this:= pushers_too_close);
		
	digital_check_and_message_init(
		object_name:= CONCAT(prc_path, '_pushers_too_close_dchk'), 
		alarm_if_input_off:= FALSE, 
		alarm_delay:= 0, 
		enabled_at_powerup:= TRUE, 
		individual_reset:= FALSE, 
		machine_reaction:= MACHINE_REACTION_EMERGENCY_STOP, 
		typology:= MESSAGE_TYPOLOGY_EMERGENCY, 
		process:= prc, 
		CONVERSION_this:= pushers_too_close_dchk);
		
	digital_check_add_boolean(
		boolean:= pushers_too_close, 
		CONVERSION_this:= pushers_too_close_dchk);
		
	process_message_init(
        object_name:= CONCAT(prc_path, '_consecutive_accumulator_reject_aem'),
        behaviour:= MESSAGE_BEHAVIOUR_STATE,
        reset_timeout:= 0,
        disableable:= TRUE,
        individual_reset:= FALSE,
        machine_reaction:= MACHINE_REACTION_STOP_IN_PHASE_ONE,
        typology:=  MESSAGE_TYPOLOGY_ABNORMAL,
        process:= prc,
        CONVERSION_this:= consecutive_accumulator_reject_asm);	
	
END_IF

IF objects_running()
THEN
	process_cycle(prc);	
	digital_check_cycle(pushers_too_close_dchk);
	
END_IF
END_ACTION

ACTION _read_process_image:
;
END_ACTION

ACTION _read_var_input:
;
END_ACTION

ACTION _set_runtime_properties:
;
END_ACTION

ACTION _write_output:
;
END_ACTION

ACTION reject:
(*************** MACHINE STATUS ***************)


IF reject_running
	AND machine_is_stop_emergency_active(csp.mch)
THEN
	reject_status_next := CSP_TRANSFER_CROSSPUSHER_REJECT_STATUS_EMERGENCY_STOP;
	process_message_set(0,0,0, csp_transfer_crosspusher_reject.remove_cartons_wem); //sets warning message, needs guards open to reset because guards have to be opened to remove the cartons
	estop_occured_in_crosspush_reject := TRUE;
ELSIF NOT machine_is_stop_emergency_active(csp.mch) //once machine is reset from the E-Stop fault, reset the estop crosspush bit
	AND reject_status = CSP_TRANSFER_CROSSPUSHER_REJECT_STATUS_EMERGENCY_STOP_FOLLOWER_MOVE
THEN
	estop_occured_in_crosspush_reject := FALSE;
END_IF
 
CASE reject_status OF
	
	CSP_TRANSFER_CROSSPUSHER_REJECT_STATUS_START:
	
		reject_done := FALSE;
				
		(* DWELL TRANSFER TO WAIT FOR CROSSPUSHER REJECT TO FINISH *)
		reject_running := TRUE;
		reject_status_next := CSP_TRANSFER_CROSSPUSHER_REJECT_STATUS_DISENGAGE_AXES;

	
	// TEMPORARILY SKIPPING	
	CSP_TRANSFER_CROSSPUSHER_REJECT_STATUS_DWELL_TRANSFER_VM:
	
		(* CHECK THAT TRANSFER IS DWELLING *)
		IF csp_transfer_virtualMaster.active_cam = DWELL_CAM
		THEN
			reject_status_next:= CSP_TRANSFER_CROSSPUSHER_REJECT_STATUS_DISENGAGE_AXES;
		END_IF
		
		
	CSP_TRANSFER_CROSSPUSHER_REJECT_STATUS_DISENGAGE_AXES:

		IF csp_transfer_crosspusher_horizontal.at_load
			AND csp_transfer_crosspusher_horizontal.axis.actual_velocity < 0.2
		THEN
			axis_stop(	
			deceleration:= csp_transfer_crosspusher_horizontal.MOTOR_MAX_DECELLERATION_DEGPS2, 
			jerk:= csp_transfer_crosspusher_horizontal.MOTOR_MAX_JERK_DEGPS3, 
			CONVERSION_this:= csp_transfer_crosspusher_horizontal.axis);
		END_IF
			
		IF ABS(csp_transfer_crosspusher_follower.axis.actual_position - csp_transfer_crosspusher_follower.slave_scaling) < 2
			AND csp_transfer_crosspusher_follower.axis.actual_velocity < 0.2
		THEN
			axis_stop(	
			deceleration:= csp_transfer_crosspusher_follower.MOTOR_MAX_DECELLERATION_DEGPS2, 
			jerk:= csp_transfer_crosspusher_follower.MOTOR_MAX_JERK_DEGPS3, 
			CONVERSION_this:= csp_transfer_crosspusher_follower.axis);
		END_IF
		
		(* DOUBLE CHECK THIS - UNSURE IF WORKING *)
		IF (csp_transfer_crosspusher_vertical.axis.actual_modulo_position < 2 OR csp_transfer_crosspusher_vertical.axis.actual_modulo_position >358)
			AND csp_transfer_crosspusher_vertical.axis.actual_velocity < 0.2
		THEN
			axis_stop(	
			deceleration:= csp_transfer_crosspusher_vertical.MOTOR_MAX_DECELLERATION_DEGPS2, 
			jerk:= csp_transfer_crosspusher_vertical.MOTOR_MAX_JERK_DEGPS3, 
			CONVERSION_this:= csp_transfer_crosspusher_vertical.axis);	
		END_IF
		
		(* VERIFY AXES ARE DISENGAGED AND STANDSTILL *)
		IF 	axis_is_standstill(csp_transfer_crosspusher_horizontal.axis)
			AND axis_is_standstill(csp_transfer_crosspusher_follower.axis)
			AND axis_is_standstill(csp_transfer_crosspusher_vertical.axis)
		THEN
			reject_status_next := CSP_TRANSFER_CROSSPUSHER_REJECT_STATUS_GEAR_FOLLOWER;
		END_IF
		
		
	CSP_TRANSFER_CROSSPUSHER_REJECT_STATUS_GEAR_FOLLOWER:
		// GEAR FOLLOWER TO CROSSPUSHER HORIZONTAL
		// CHECK GEAR
		// ADVANCE		
		(* GEAR FOLLOWER TO HORIZONTAL *)
		axis_engage_position_gear(
			ratio:= -1, 
			acceleration:= csp_transfer_crosspusher_follower.MOTOR_MAX_ACCELLERATION_DEGPS2/4, 
			deceleration:= csp_transfer_crosspusher_follower.MOTOR_MAX_DECELLERATION_DEGPS2/4, 
			jerk:= csp_transfer_crosspusher_follower.MOTOR_MAX_JERK_DEGPS3, 
			master:= csp_transfer_crosspusher_horizontal.axis, 
			CONVERSION_this:= csp_transfer_crosspusher_follower.axis);
			
		(* CHECK GEAR AND ADVANCE *)
		IF axis_is_gear_engaged(csp_transfer_crosspusher_follower.axis)
		THEN
			reject_status_next := CSP_TRANSFER_CROSSPUSHER_REJECT_STATUS_MOVE_TO_REJECT_POS;
		END_IF

		
	CSP_TRANSFER_CROSSPUSHER_REJECT_STATUS_MOVE_TO_REJECT_POS:
	
		// MOVE CROSSSPUSHER HORIZONTAL TO REJECT POSITION - check
		// ADVANCE ON STANDSTILL - check
		(* MOVE CORRPUSHER HORIZONTAL TO REJECT POSITION *)
		(* VERIFY LOADER IS CLEAR *)
		IF csp_transfer_crosspusher.loader_clear
			AND NOT digital_actuator_is_active(csp_transfer_crosspusher_reject.reject_sact)
			//AND csp_case_loader_virtualMaster.active_cam = DWELL_CAM
		THEN
			axis_move_absolute(
			position:= horizontal_reject_position, 
			velocity:= reject_velocity, 
			direction:= AXIS_SHORTEST_WAY, 
			acceleration:= csp_transfer_crosspusher_horizontal.MOTOR_MAX_ACCELLERATION_DEGPS2/2, 
			deceleration:= csp_transfer_crosspusher_horizontal.MOTOR_MAX_DECELLERATION_DEGPS2/2, 
			jerk:= csp_transfer_crosspusher_horizontal.MOTOR_MAX_JERK_DEGPS3, 
			buffer_mode:= AXIS_BUFFER_MODE_ABORTING, 
			CONVERSION_this:= csp_transfer_crosspusher_horizontal.axis);
		END_IF
			
		(* CHECK THAT AXIS IS MOVING TO REJECT - ADVANCE *)
		IF axis_is_absolute_moving(csp_transfer_crosspusher_horizontal.axis)
		THEN
			reject_status_next := CSP_TRANSFER_CROSSPUSHER_REJECT_STATUS_VERIFY_HORIZONTAL_POS;
		END_IF

		
	CSP_TRANSFER_CROSSPUSHER_REJECT_STATUS_VERIFY_HORIZONTAL_POS:
	
		// CHECK HORIZONTAL IS WITHIN REJECT POSITION PHASE WINDOW - check
		// CHECK THAT FOLLOWER IS WITHIN REJECT POSITION PHASE WINDOW
		// ADVANCE - check
		IF csp_transfer_crosspusher_horizontal.axis.actual_position < crosspusher_horiz_at_reject_high_limit			
			AND csp_transfer_crosspusher_horizontal.axis.actual_position > crosspusher_horiz_at_reject_low_limit	
			AND axis_is_standstill(csp_transfer_crosspusher_horizontal.axis)
		THEN
			reject_status_next := CSP_TRANSFER_CROSSPUSHER_REJECT_STATUS_UNGEAR_FOLLOWER;
		END_IF
		
	
	CSP_TRANSFER_CROSSPUSHER_REJECT_STATUS_UNGEAR_FOLLOWER:
		
		(* BREAK GEAR ON FOLLOWER *)	
		IF axis_is_gear_engaged(csp_transfer_crosspusher_follower.axis)
		THEN
			axis_stop(	
				deceleration:= csp_transfer_crosspusher_follower.MOTOR_MAX_DECELLERATION_DEGPS2, 
				jerk:= csp_transfer_crosspusher_follower.MOTOR_MAX_JERK_DEGPS3, 
				CONVERSION_this:= csp_transfer_crosspusher_follower.axis);
		END_IF
	
		(* CHECK NOT GEARED - ADVANCE *)
		IF axis_is_standstill(csp_transfer_crosspusher_follower.axis)
		THEN
			reject_status_next := CSP_TRANSFER_CROSSPUSHER_REJECT_STATUS_MOVE_FOLLOWER;
		END_IF
		
		
	CSP_TRANSFER_CROSSPUSHER_REJECT_STATUS_MOVE_FOLLOWER:
		
		(* MOVE CORRPUSHER HORIZONTAL TO REJECT POSITION *)
		IF csp_transfer_crosspusher.loader_clear
		THEN
			axis_move_absolute(
				position:= follower_reject_position, 
				velocity:= reject_velocity, 
				direction:= AXIS_NEGATIVE_DIRECTION, 
				acceleration:= csp_transfer_crosspusher_horizontal.MOTOR_MAX_ACCELLERATION_DEGPS2/2, 
				deceleration:= csp_transfer_crosspusher_horizontal.MOTOR_MAX_DECELLERATION_DEGPS2/2, 
				jerk:= csp_transfer_crosspusher_horizontal.MOTOR_MAX_JERK_DEGPS3, 
				buffer_mode:= AXIS_BUFFER_MODE_ABORTING, 
				CONVERSION_this:= csp_transfer_crosspusher_follower.axis);
		END_IF
		
		(* CHECK THAT AXIS IS MOVING TO REJECT - ADVANCE *)
		IF axis_is_absolute_moving(csp_transfer_crosspusher_follower.axis)
		THEN
			reject_status_next := CSP_TRANSFER_CROSSPUSHER_REJECT_STATUS_VERIFY_FOLLOWER_POS;
		END_IF
		
		
	CSP_TRANSFER_CROSSPUSHER_REJECT_STATUS_VERIFY_FOLLOWER_POS:
		
		IF csp_transfer_crosspusher_follower.axis.actual_position < crosspusher_foll_at_reject_high_limit			
			AND csp_transfer_crosspusher_follower.axis.actual_position > crosspusher_foll_at_reject_low_limit	
			AND axis_is_standstill(csp_transfer_crosspusher_follower.axis)
		THEN
			reject_status_next := CSP_TRANSFER_CROSSPUSHER_REJECT_STATUS_REJECT_STACK;
		END_IF
		
	
	CSP_TRANSFER_CROSSPUSHER_REJECT_STATUS_REJECT_STACK:
	
	// BEGIN REJECT OF STACK USING csp_transfer_crosspusher_reject PROGRAM
	// WAIT FOR REJECT EXTENSION AND ADVANCE
		IF csp_transfer_crosspusher_reject.reject_status > 0
		THEN
			reject_status_next := CSP_TRANSFER_CROSSPUSHER_REJECT_STATUS_VERIFY;
		END_IF
	
		
	CSP_TRANSFER_CROSSPUSHER_REJECT_STATUS_VERIFY:
	
		IF csp_transfer_crosspusher_reject.reject_complete 
			AND digital_actuator_is_inactive(csp_transfer_crosspusher_reject.reject_sact)
		THEN
			reject_status_next := CSP_TRANSFER_CROSSPUSHER_REJECT_STATUS_RETURN_HORIZONTAL;
		END_IF
		//TODO return follower to previous position and regear
	

	CSP_TRANSFER_CROSSPUSHER_REJECT_STATUS_RETURN_HORIZONTAL:
	
		// CALCULATE CROSSPUSHER HORIZONTAL POSITION BASED ON TRANSFER VIRTUAL MASTER - check
		// ABSOLUTE MOVE TO POSITION - check
		// ON AXIS MOVING, ADVANCE - check
		axis_move_absolute(
			position:= csp_transfer_crosspusher_horizontal.load_position, 
			velocity:= reject_velocity, 
			direction:= AXIS_SHORTEST_WAY, 
			acceleration:= csp_transfer_crosspusher_horizontal.MOTOR_MAX_ACCELLERATION_DEGPS2/2, 
			deceleration:= csp_transfer_crosspusher_horizontal.MOTOR_MAX_DECELLERATION_DEGPS2/2, 
			jerk:= csp_transfer_crosspusher_horizontal.MOTOR_MAX_JERK_DEGPS3, 
			buffer_mode:= AXIS_BUFFER_MODE_ABORTING, 
			CONVERSION_this:= csp_transfer_crosspusher_horizontal.axis);
	
		IF axis_is_absolute_moving(csp_transfer_crosspusher_horizontal.axis)
		THEN
			reject_status_next := CSP_TRANSFER_CROSSPUSHER_REJECT_STATUS_HORIZONTAL_RETURNING;
		END_IF	
	
	
	CSP_TRANSFER_CROSSPUSHER_REJECT_STATUS_HORIZONTAL_RETURNING:
		
		IF axis_is_absolute_moving(csp_transfer_crosspusher_horizontal.axis)
		THEN
			reject_status_next := CSP_TRANSFER_CROSSPUSHER_REJECT_STATUS_RETURN_FOLLOWER;
		END_IF

		
	CSP_TRANSFER_CROSSPUSHER_REJECT_STATUS_RETURN_FOLLOWER:
		
		IF csp_transfer_crosspusher.loader_clear
			AND NOT digital_actuator_is_active(csp_transfer_crosspusher_reject.reject_sact)
		THEN
			axis_move_absolute(
				position:= csp_transfer_crosspusher_follower.slave_scaling, 
				velocity:= reject_velocity, 
				direction:= AXIS_SHORTEST_WAY, 
				acceleration:= csp_transfer_crosspusher_follower.MOTOR_MAX_ACCELLERATION_DEGPS2/4, 
				deceleration:= csp_transfer_crosspusher_follower.MOTOR_MAX_DECELLERATION_DEGPS2/4, 
				jerk:= csp_transfer_crosspusher_follower.MOTOR_MAX_JERK_DEGPS3, 
				buffer_mode:= AXIS_BUFFER_MODE_ABORTING, 
				CONVERSION_this:= csp_transfer_crosspusher_follower.axis);
		END_IF
	
		IF axis_is_absolute_moving(csp_transfer_crosspusher_follower.axis)
		THEN
			reject_status_next := CSP_TRANSFER_CROSSPUSHER_REJECT_STATUS_FOLLOWER_RETURNING;
		END_IF	
		
		
	CSP_TRANSFER_CROSSPUSHER_REJECT_STATUS_FOLLOWER_RETURNING:
		
		IF axis_is_absolute_moving(csp_transfer_crosspusher_follower.axis)
		THEN
			reject_status_next := CSP_TRANSFER_CROSSPUSHER_REJECT_STATUS_VERIFY_AT_LOAD;
		END_IF
	
	
	CSP_TRANSFER_CROSSPUSHER_REJECT_STATUS_VERIFY_AT_LOAD:
	
		IF axis_is_standstill(csp_transfer_crosspusher_horizontal.axis)
			AND csp_transfer_crosspusher_horizontal.at_load//csp_transfer_crosspusher_horizontal.axis.actual_position < crosspusher_horiz_at_load_high_limit
			AND axis_is_standstill(csp_transfer_crosspusher_follower.axis)
			AND ABS(csp_transfer_crosspusher_follower.axis.actual_position - csp_transfer_crosspusher_follower.slave_scaling) < 2 //axis.actual_position < crosspusher_foll_at_reject_high_limit
		THEN
			reject_status_next := CSP_TRANSFER_CROSSPUSHER_REJECT_STATUS_RUN_AXES;
		END_IF
	
	
	CSP_TRANSFER_CROSSPUSHER_REJECT_STATUS_RUN_AXES:
	
		// TESTING
		reject_run_transfer := FALSE;
		reject_running := FALSE;
		reject_done := TRUE;
		
		IF 	axis_is_cam_engaged(csp_transfer_crosspusher_horizontal.axis)
			AND axis_is_cam_engaged(csp_transfer_crosspusher_follower.axis)
			AND axis_is_cam_engaged(csp_transfer_crosspusher_vertical.axis)
		THEN
			reject_status_next := CSP_TRANSFER_CROSSPUSHER_REJECT_STATUS_DONE;
		END_IF
		
		
	CSP_TRANSFER_CROSSPUSHER_REJECT_STATUS_DONE:
	
		// TESTING
		reject_dwell_transfer := FALSE;
		
		IF csp_transfer_virtualMaster.active_cam = FORWARD_CAM
		THEN
			reject_status_next := CSP_TRANSFER_CROSSPUSHER_REJECT_STATUS_WAITING;
		END_IF
		
		
	CSP_TRANSFER_CROSSPUSHER_REJECT_STATUS_WAITING:
	
		;
		
		
	CSP_TRANSFER_CROSSPUSHER_REJECT_STATUS_EMERGENCY_STOP:
	
		IF machine_is_running(csp.mch)
		THEN
			reject_status_next := CSP_TRANSFER_CROSSPUSHER_REJECT_STATUS_EMERGENCY_STOP_ENABLE;
		END_IF
		

	CSP_TRANSFER_CROSSPUSHER_REJECT_STATUS_EMERGENCY_STOP_ENABLE:
	
		axis_enable(csp_transfer_crosspusher_horizontal.axis);
		axis_enable(csp_transfer_crosspusher_follower.axis);
		
		IF 	axis_is_enabled(csp_transfer_crosspusher_horizontal.axis)
			AND axis_is_enabled(csp_transfer_crosspusher_follower.axis)
		THEN
			reject_status_next := CSP_TRANSFER_CROSSPUSHER_REJECT_STATUS_EMERGENCY_STOP_GOTO;
		END_IF
		
		
	CSP_TRANSFER_CROSSPUSHER_REJECT_STATUS_EMERGENCY_STOP_GOTO:
	
		(* HAS NOT REJECTED STACK - PHASE THE FOLLOWER TO IT'S POSITION AND REGEAR *)
		IF 	reject_status_last_state <= CSP_TRANSFER_CROSSPUSHER_REJECT_STATUS_VERIFY
			AND csp_transfer_crosspusher.loader_clear
			AND NOT digital_actuator_is_active(csp_transfer_crosspusher_reject.reject_sact)
		THEN			
			(*IF csp_transfer_crosspusher_horizontal.axis.actual_position < 0
			THEN
				follower_calc_pos := follower_pos_if_horiz_is_neg;
			ELSE
				follower_calc_pos := calc_distance_between_pushers; // +40 added to fix bug with follower going wrong way
			END_IF	*)
			
			IF calc_adjustment_for_follower > 0
			THEN
				follower_calc_pos := csp_transfer_crosspusher_follower.axis.actual_position - ABS(calc_adjustment_for_follower);
			ELSE
				follower_calc_pos := csp_transfer_crosspusher_follower.axis.actual_position + ABS(calc_adjustment_for_follower);
			END_IF	
			
			(* VERIFIES CALCULATED POS IS NOT ABOVE 850 *)
			IF follower_calc_pos > 850 (* HARD CODED INDRAWORKS VALUE IS 865 BUT 850 IS USED FOR A SAFE POSITION *)
			THEN
				follower_calc_pos := 850;
			END_IF
					
			(* MOVE FOLLOWER TO CORRECT POSITION FROM HORIZONTAL *)
			axis_move_absolute(
				position:= follower_calc_pos, 
				velocity:= reject_velocity, 
				direction:= AXIS_SHORTEST_WAY, 
				acceleration:= csp_transfer_crosspusher_follower.MOTOR_MAX_ACCELLERATION_DEGPS2/4, 
				deceleration:= csp_transfer_crosspusher_follower.MOTOR_MAX_DECELLERATION_DEGPS2/4, 
				jerk:= csp_transfer_crosspusher_follower.MOTOR_MAX_JERK_DEGPS3, 
				buffer_mode:= AXIS_BUFFER_MODE_ABORTING, 
				CONVERSION_this:= csp_transfer_crosspusher_follower.axis);
				
			IF axis_is_absolute_moving(csp_transfer_crosspusher_follower.axis)
			THEN
				reject_status_next := CSP_TRANSFER_CROSSPUSHER_REJECT_STATUS_EMERGENCY_STOP_FOLLOWER_MOVE;
			END_IF
					
		(* REJECT COMPLETED - PHASE AXES BACK TO LOAD *)
		ELSIF reject_status_last_state > CSP_TRANSFER_CROSSPUSHER_REJECT_STATUS_VERIFY
		THEN
			reject_status_next := CSP_TRANSFER_CROSSPUSHER_REJECT_STATUS_RETURN_HORIZONTAL;
		END_IF
		
		
	CSP_TRANSFER_CROSSPUSHER_REJECT_STATUS_EMERGENCY_STOP_FOLLOWER_MOVE:
		
		IF axis_is_standstill(csp_transfer_crosspusher_follower.axis)
		THEN
			reject_status_next := CSP_TRANSFER_CROSSPUSHER_REJECT_STATUS_GEAR_FOLLOWER;
		END_IF		
END_CASE


IF 	NOT debug_state_machine
	OR
	debug_reject_machine_one_step	
THEN
	reject_status := reject_status_next;
	debug_reject_machine_one_step := FALSE;
END_IF

(* Connection timeout *)
IF	reject_running
THEN
	IF	timer_is_expired(reject_time_out_tmr)
	THEN
		//process_message_set(1, reject_status, 0, reject_faulted_aem);
	END_IF
ELSE
	timer_restart(20000, reject_time_out_tmr);
END_IF
END_ACTION

END_PROGRAM

// ---- Application/CSP/Transfer/Crosspusher/Follower/csp_transfer_crosspusher_follower.TcPOU
(*********************************** G.D S.p.A. - Technical Department ***********************************
============= PROGRAM INFO ============
FOLDER:             TBD
MACHINES INVOLVED:  TBD 

============= DESCRIPTION =============
csp machine declaration

============= REVISIONS ===============
Date		Version	 	Author      	Description             
----------	-------		------------  	--------------------------------------------
2019/04/05 	0000.00	 	M.Grasso		Creation of the PRG

**********************************************************************************************************)
(*$R process_ref := prc; $*)
PROGRAM csp_transfer_crosspusher_follower
VAR
	
	prc:												process;
	prc_path:											STRING;
	
	axis:												axis;
	
	phase_velocity_degps:								LREAL := 250.0;
		
	home_position_master_offset_deg:					LREAL := 0;
	axis_calculate_cam_slave_master_position_deg:		LREAL := 0.0;
	axis_calculated_cam_slave_position_deg:				LREAL := 0.0;	
	slave_position_has_been_calculated:					BOOL  := FALSE;
	
	engage_enable:										BOOL := TRUE;
	
	slave_scaling:										LREAL := 350; (*$P $*)
	master_scaling:										LREAL := 1;
	
	slave_scale_test:									LREAL;
	
	master_offset:										LREAL := 0;
	master_offset_phase:								LREAL;
	master_engage_mode:									axis_cam_engage_mode_enum;
	slave_offset:										LREAL := 0;
	slave_offset_input:									LREAL := 0;
	
	engage_mode:										axis_cam_engage_mode_enum;
	
	dwell:												BOOL;
	load_to_upstack_to_load:							BOOL;
	
	dwell_test:											BOOL;
	load_to_upstack_to_load_test:						BOOL;
	
	active_cam:											DINT := DWELL_CAM;
	next_cam:											DINT := DWELL_CAM;
	
	connection_status: 									csp_transfer_crosspusher_connection_status_enum;
	connection_status_next: 							csp_transfer_crosspusher_connection_status_enum;
	connection_done: 									BOOL;
	connection_running: 								BOOL;
	connection_error:									BOOL;
	connection_time_out_tmr:							timer;
	connection_faulted_aem:	 							message;
	connection_conditions:								BOOL;
	connection_done_motcond:							motorization_conditioner;
	connection_motorization_moving:						BOOL;
	
	next_activation_position:							LREAL;	
	activation_position:								LREAL := 0.0;
	
	phase_delay_tmr:									timer;
	phase_delay:										UDINT := 1000;
	
	phase_status: 										csp_transfer_crosspusher_phase_status_enum;
	phase_status_next: 									csp_transfer_crosspusher_phase_status_enum;
	phase_done: 										BOOL;
	phase_running: 										BOOL;
	phase_error:										BOOL;
	phase_time_out_tmr:									timer;
	phase_faulted_aem:	 								message;
	phase_conditions:									BOOL;
	phase_slave_position:								LREAL;
	
	
	disable_req:										BOOL;
	debug_phase_state_machine:							BOOL := FALSE;
	debug_phase_machine_one_step:						BOOL := FALSE;
	debug_connection_state_machine:						BOOL := FALSE;
	debug_connection_machine_one_step:					BOOL := FALSE;
	debug_immediate_stop_aem:							message;
	debug_immediate_stop:								BOOL;
	
	torque_limit:										INT := 500; (*$P $*)
	torque_limit_old:									INT;
	
	direction_fwd:										BOOL;
	
	in_accu_safe_pos:                                   BOOL := FALSE;
    accu_tolerance:                                     INT := 5;
    accu_safe_pos:                                      INT;	(*$P $*)
	
	servo_on_condition: 								BOOL;
	enable_delay: TON;
	Torque_force_constant: 								LREAL := 1.33;
END_VAR

VAR CONSTANT
	MOTOR_MAX_VELOCITY_DEGPS:							LREAL := 9600;
	MOTOR_MAX_ACCELLERATION_DEGPS2:						LREAL := 9600;
	MOTOR_MAX_DECELLERATION_DEGPS2:						LREAL := 9600;
	MOTOR_MAX_JERK_DEGPS3:								LREAL := 100000000; 
	MOTOR_MAX_FOLLOWING_ERROR_DEG:						LREAL := 2;
	
END_VAR

_read_var_input();

_object_manager();

IF NOT objects_running()
THEN
	RETURN;	
END_IF

_read_process_image();

_mode_manager();

CASE process_get_mode(prc) OF
	MODE_ABSENT:
		IF axis_get_mode(axis) = MODE_TEST
		THEN
			safety_integrated_series_close(csp_transfer_main_safety_drives_SD41500.chA_smes_sis);
		END_IF
		RETURN;
	MODE_INACTIVE:
		RETURN;
	MODE_TEST:
		_handle_process_test();
END_CASE

(********************************* BODY *********************************)
axis.actual_torque := (axis.actual_current * Torque_force_constant)/1000;

(* Acc-U-Change Safe Position *)
accu_safe_pos := LREAL_TO_INT(slave_scaling);

IF 	ABS(axis.actual_position - accu_safe_pos)  < accu_tolerance
	OR (360 - axis.actual_position) < accu_tolerance
THEN
	in_accu_safe_pos := TRUE;
ELSE
	in_accu_safe_pos := FALSE;   
END_IF

(* Sets torque Limit *)
IF torque_limit <> torque_limit_old
THEN
	IF soe_drive_channel_write_parameter(
		channel:= csp_transfer_crosspusher_follower.axis.soe_drive_channel, 
		idn:= S_0_IDN + 92, 
		data_element:= soe_drive_element_value, 
		data_source:= ADR(torque_limit), 
		data_lenght:= SIZEOF(torque_limit),
		CONVERSION_this:= csp_transfer_crosspusher_follower.axis.soe_drive^) = SOE_DRIVE_RETURN_VALUE_DONE
	THEN
		torque_limit_old := torque_limit;
	END_IF
END_IF

IF machine_is_stopped(csp.mch)
THEN
	phase_error := FALSE;
	connection_error := FALSE;
END_IF

(* SLAVE SCALING BY CASE DIMENSIONS *)
slave_scaling := 	(
						csp_main_brand.carton_dimension.carton_size_L_mm 
						* 
						csp_main_brand.case_pattern.case_pattern_L
					) 
					+ 
					csp_transfer_crosspusher.horiz_to_follower_diff 
					+ 
					csp_transfer_crosspusher.horiz_to_follower_tolerance;

(* Connection Done MOT COND *)
IF connection_done
THEN 
	motorization_conditioner_start_done(connection_done_motcond);
END_IF

(* SENDS TO SPECIFIC STATE IF REJECT RUNNING *)
IF csp_transfer_crosspusher.reject_running
THEN
	connection_status_next := CSP_TRANSFER_CROSSPUSHER_STATUS_CONNECTION_WAIT_REJECT;
END_IF

(* CHECK WHAT CAM TO RUN ON PHASE EDGE *)
IF phase_edge(csp_transfer_crosspusher_virtualMaster.cam_change_check_ph) (* CROSSPUSHER VIRTUAL AT CHECK PHASE DEG *)
	AND connection_status = CSP_TRANSFER_CROSSPUSHER_STATUS_CONNECTION_CHECK_CHANGE_CAM
THEN
	(* LOGIC TO DETERMINE IF RUN TO LOAD *)
	IF load_to_upstack_to_load_test (* TEST BIT *)
		OR
		(
		csp_transfer_upstacker.stack_made (* UPSTACKER MADE CORRECT AMOUNT OF STACK *)
		AND csp_transfer_crosspusher_horizontal.at_upstack (* VERIFIES THE HORIZONTAL IS AT THE UPSTACKER BEFORE RUNNING *)
		AND NOT csp_transfer_upstacker.stack_at_loader (* MAKES SURE A STACK IS NOT ALREADY AT THE LOADER *)
		)
	THEN
		load_to_upstack_to_load := TRUE;
	(* CONDITIONS NOT MET - DWELL *)
	ELSE
		dwell := TRUE;
	END_IF
	
END_IF

(* DWELL CAM BECAUSE LOADER NOT CLEAR - IMMEDIATELY *)
(* Used to immediately queue dwell given the Follower will always dwell after move *)
IF 	active_cam = TRANSFER_CROSSPUSHER_FOLLOWER_TO_UPSTACK_TO_LOAD
	AND csp_transfer_crosspusher.loader_status = csp_transfer_crosspusher_loader_clear_status.NOT_CLEAR 
THEN
	connection_status_next := CSP_TRANSFER_CROSSPUSHER_STATUS_CONNECTION_IMMEDIATE_CHANGE;
	connection_status := CSP_TRANSFER_CROSSPUSHER_STATUS_CONNECTION_IMMEDIATE_CHANGE;
END_IF

(* REWRITES ACTIVE CAM IF BECOMES 0 *)
IF active_cam = 0
THEN 
	active_cam := DWELL_CAM;
END_IF

(* CLEARS CONNECTION AND PHASE ERRORS *)
IF machine_is_stopped(csp.mch)
	OR machine_is_stop_emergency_active(csp.mch)
	OR machine_is_ready(csp.mch)
	OR csp_main_services_pushbuttons.i_reset_button
THEN
	connection_error := FALSE;
	phase_error := FALSE;
END_IF

(* RESETS AXES IF PHASE DONE AND CONNECTION DONE AND DISABLED *)
IF phase_done
	AND connection_done
	AND axis_is_disabled(axis)
THEN
	phase_done := FALSE;
	connection_done := FALSE;
END_IF

(* TELLS THE FOLLOWER WHAT THE PROFILE SHOULD BE ON A CLEARED LOAD *)
IF csp_transfer_upstacker.stack_removed_from_upstack
	OR message_is_on(csp_transfer_crosspusher.pushers_too_close_dchk.alarm_asm.message)
	OR csp_transfer_crosspusher.reject_running
THEN
	active_cam := DWELL_CAM;
	next_cam := DWELL_CAM;
END_IF

(* RUNS ACTIONS FOR AXIS *)
phase();
connection();
_set_runtime_properties();

(************************************************************************)

_handle_messages();

_write_output();

ACTION _handle_messages:
;
END_ACTION

ACTION _handle_process_test:
;
END_ACTION

ACTION _mode_manager:
IF process_mode_req_is_pending(prc)
THEN
    process_apply_mode_req_first_step(prc);
    CASE process_get_mode(prc) OF
        MODE_TO_ABSENT:
			;
        MODE_TO_INACTIVE:
			;
        MODE_TO_TEST:
			;
        MODE_TO_OPERATIONAL:
			;
    END_CASE
    process_apply_mode_req_second_step(prc);
END_IF
END_ACTION

ACTION _object_manager:
IF objects_initialization()
THEN
	sub_process_init(
		object_name								:= 'csp_transfer_crosspusher_follower.prc', 
		process									:= csp_transfer_crosspusher.prc, 
		CONVERSION_this							:= prc);
		
	prc_path 									:= process_get_path(prc);
	
	(* AXIS INIT *)
	axis_init(
		object_name								:= CONCAT(prc_path, '_axis'), 
		axis_type								:= AXIS_TYPE_SERVO, 
		encoder_scaling_factor					:= G_SERVO_ENCODER_SCALING_FACTOR_DEGPINC,
		modulo									:= G_NO_MODULO_DEG, 
		process									:= prc, 
		CONVERSION_this							:= axis);
		
	axis_init_absolute_encoder_preset(
		position								:= 645.2, 
		CONVERSION_this							:= axis);
	
	axis_set_max_dynamic(
		reference_velocity						:=	MOTOR_MAX_VELOCITY_DEGPS,
		velocity								:=	MOTOR_MAX_VELOCITY_DEGPS,
		acceleration							:=	MOTOR_MAX_ACCELLERATION_DEGPS2,
		deceleration							:=	MOTOR_MAX_DECELLERATION_DEGPS2,
		jerk									:=	MOTOR_MAX_JERK_DEGPS3,
		following_error							:=	MOTOR_MAX_FOLLOWING_ERROR_DEG,
		CONVERSION_this							:=	axis);
		
	(* AXIS SAFETY *)
	axis_add_soe_drive(
		channel									:=	SOE_DRIVE_CHANNEL_A,
		soe_drive								:=	csp_transfer_main_drives.SD41500_drv,
		CONVERSION_this							:=	axis);
		
	axis_add_safety_integrated_series(
		safety_integrated_series 				:= csp_transfer_main_safety_drives_SD41500.chA_smes_sis,
		CONVERSION_this							:= axis);
	
		
	(* DEBUG MESSAGE *)	
	process_message_init(
		object_name								:=	CONCAT(prc_path, 'debug_immediate_stop_aem'), 
		behaviour								:=	MESSAGE_BEHAVIOUR_STATE,
		reset_timeout							:=	0,
		disableable								:=	TRUE,
		individual_reset						:=	FALSE,
		machine_reaction						:=	MACHINE_REACTION_NORMAL_STOP,
		typology								:=	MESSAGE_TYPOLOGY_ABNORMAL,
		process									:=	prc,
		CONVERSION_this							:=	debug_immediate_stop_aem);	
		
		
	(* PHASE MESSAGES *)
	process_message_init(
		object_name								:=	CONCAT(prc_path, '_phase_faulted_aem'), 
		behaviour								:=	MESSAGE_BEHAVIOUR_EVENT,
		reset_timeout							:=	0,
		disableable								:=	TRUE,
		individual_reset						:=	FALSE,
		machine_reaction						:=	MACHINE_REACTION_NORMAL_STOP,
		typology								:=	MESSAGE_TYPOLOGY_ABNORMAL,
		process									:=	prc,
		CONVERSION_this							:=	phase_faulted_aem);
	
	timer_init(
		object_name								:= CONCAT(prc_path, 'phase_time_out_tmr'),
		process									:= prc,
		CONVERSION_this							:= phase_time_out_tmr);
		
	timer_init(
		object_name								:= CONCAT(prc_path, 'phase_delay_tmr'),
		process									:= prc,
		CONVERSION_this							:= phase_delay_tmr);
		
	(* CONNECTION MESSAGES *)
	process_message_init(
		object_name								:=	CONCAT(prc_path, '_connection_faulted_aem'), 
		behaviour								:=	MESSAGE_BEHAVIOUR_EVENT,
		reset_timeout							:=	0,
		disableable								:=	TRUE,
		individual_reset						:=	FALSE,
		machine_reaction						:=	MACHINE_REACTION_NORMAL_STOP,
		typology								:=	MESSAGE_TYPOLOGY_ABNORMAL,
		process									:=	prc,
		CONVERSION_this							:=	connection_faulted_aem);
		
	timer_init(
		object_name								:= CONCAT(prc_path, 'connection_time_out_tmr'),
		process									:= prc,
		CONVERSION_this							:= connection_time_out_tmr);
		
	motorization_conditioner_init(
		object_name								:=	CONCAT(prc_path, 'connection_done_motcond'),
		velocity_limit							:=	0.0,
		velocity_limit_active					:=	FALSE,
		idle_handshake_active					:=	FALSE,
		execute_handshake_active				:=	TRUE,
		hold_handshake_active					:=	FALSE,
		suspend_handshake_active				:=	FALSE,
		complete_handshake_active				:=	FALSE,
		abort_handshake_active					:=	FALSE,
		stop_handshake_active					:=	FALSE,
		origin									:=	MOTORIZATION_CONDITIONER_ORIGIN_INTERNAL,
		manager									:=	csp_main_motorization_manager.motm,
		process									:=	prc,
		CONVERSION_this							:=	connection_done_motcond);
	
	jog_manager_add_axis(
		list_index								:= SMTR41503_TRANSFER_CROSSPUSHER_FOLLOWER,
		axis									:= axis,
		master_axis								:= FALSE,
		jog_type								:= JOG_TYPE_LINEAR,
		sw_limit_positive						:= 850,
		sw_limit_negative						:= -20,
		CONVERSION_this							:= csp_main_jogManager.jog_manager_real);		
		
		
END_IF

IF objects_running()
THEN
	process_cycle(prc);	
	axis_cycle(axis);		
	motorization_conditioner_cycle(connection_done_motcond);	
END_IF
END_ACTION

ACTION _read_process_image:
;
END_ACTION

ACTION _read_var_input:
;
END_ACTION

ACTION _set_runtime_properties:
(* Cam management *)
IF 	connection_done
THEN
	active_cam := axis.engaged_cam.cam_id;
END_IF

enable_delay(IN:=axis_is_ready_to_enable(axis) , PT:=T#2S , Q=> servo_on_condition , ET=> );
END_ACTION

ACTION _write_output:
;
END_ACTION

ACTION connection:
connection_conditions :=	
	axis_is_ok(FALSE, axis)
	AND
	servo_on_condition
	AND
	NOT process_message_is_on(connection_faulted_aem)
	AND
	phase_done;

(* connection_done reset *)
IF	connection_done
	AND	
	NOT connection_conditions
	AND
	NOT csp.o_machine_is_running
THEN
	connection_done := FALSE;
END_IF

(* Exit conditions *)
IF	NOT connection_conditions 
	AND
	NOT motorization_manager_is_stopping(csp_main_motorization_manager.motm)	
THEN	
	connection_status_next := CSP_TRANSFER_CROSSPUSHER_STATUS_CONNECTION_ERROR;
	connection_status := connection_status_next;	
END_IF

(*************** MACHINE STATUS ***************)
CASE connection_status OF

	CSP_TRANSFER_CROSSPUSHER_STATUS_CONNECTION_START:	(* Start connection *)
	
		IF	motorization_manager_is_starting(csp_main_motorization_manager.motm) //TODOPZ: da decidere a che livello usare le variabili di i e o: wn_feeding.i_motorization_is_starting?					
		THEN
			connection_running := TRUE;
			connection_status_next := CSP_TRANSFER_CROSSPUSHER_STATUS_CONNECTION_ENGAGE;
		END_IF
		
		
	CSP_TRANSFER_CROSSPUSHER_STATUS_CONNECTION_ENGAGE:		
			
		IF active_cam = TRANSFER_CROSSPUSHER_FOLLOWER_TO_UPSTACK_TO_LOAD
		THEN
			engage_mode := AXIS_CAM_ENGAGE_ABSOLUTE;
			slave_offset := slave_offset_input;
			master_engage_mode := AXIS_CAM_ENGAGE_RELATIVE;
			master_offset_phase := csp_transfer_crosspusher_virtualMaster.axis.actual_modulo_position;
		ELSIF active_cam = DWELL_CAM
		THEN
			engage_mode := AXIS_CAM_ENGAGE_RELATIVE;
			slave_offset := 0;
			master_engage_mode := AXIS_CAM_ENGAGE_ABSOLUTE;
			master_offset_phase := 0.0;
		END_IF
			
		axis_engage_cam(
			cam_id							:=	active_cam,	
			master_engage_mode				:=	master_engage_mode,
			slave_engage_mode				:=	engage_mode,
			activation_mode					:=	AXIS_CAM_ACTIVATION_IMMEDIATELY,
			activation_position				:=	0.0,
			master_scaling_mode				:=	AXIS_CAM_SCALING_MODE_USER_DEFINED,
			slave_scaling_mode				:=	AXIS_CAM_SCALING_MODE_USER_DEFINED,
			master_offset					:=	master_offset + master_offset_phase,
			slave_offset					:=	slave_offset,
			master_scaling					:=	master_scaling,
			slave_scaling					:=	slave_scaling,
			interpolation_type				:=	AXIS_CAM_INTERPOLATION_SPLINE,	 
			master							:=	csp_transfer_crosspusher_virtualMaster.axis,
			CONVERSION_this					:=	axis);
		
		connection_status_next:= CSP_TRANSFER_CROSSPUSHER_STATUS_CONNECTION_ENGAGED;
	
		
	CSP_TRANSFER_CROSSPUSHER_STATUS_CONNECTION_ENGAGED:
	
		IF 	axis_is_cam_engaged(axis) 
		THEN				
			IF	active_cam <> next_cam
			THEN							
				connection_status_next := CSP_TRANSFER_CROSSPUSHER_STATUS_CONNECTION_CHANGE_CAM;
			ELSE
				connection_status_next:= CSP_TRANSFER_CROSSPUSHER_STATUS_CONNECTION_DONE;
			END_IF
		END_IF
		
		
	CSP_TRANSFER_CROSSPUSHER_STATUS_CONNECTION_CHECK_CHANGE_CAM:						
		
		(* DWELL - ALWAYS TAKES PLACE AT LOAD POSITION *)
		IF dwell
		THEN 		
			CASE active_cam OF
				
				DWELL_CAM:
					dwell := FALSE;

				TRANSFER_CROSSPUSHER_FOLLOWER_TO_UPSTACK_TO_LOAD:
					dwell := FALSE;	 
					next_cam := DWELL_CAM;					
			END_CASE			
		END_IF
			
		(* FROM LOAD POSITION TO UPSTACKER POSITION *)
		IF load_to_upstack_to_load
			AND (
					(* USED FOR 2 STACK TO QUEUE MOVE TO LOAD *)
					(csp_main_brand.case_pattern.case_pattern_W = 2
					AND csp_transfer_virtualMaster.section_0_180) (* PHASE CHECK BASED OFF OF STACK COUNT *)
				OR 
					(* USED FOR 3 STACK TO QUEUE MOVE TO LOAD *)
					(csp_main_brand.case_pattern.case_pattern_W = 3
					AND csp_transfer_virtualMaster.section_120_240)
				)
		THEN			
			CASE active_cam OF
			
				DWELL_CAM:
					load_to_upstack_to_load := FALSE;
					next_cam := TRANSFER_CROSSPUSHER_FOLLOWER_TO_UPSTACK_TO_LOAD;

				TRANSFER_CROSSPUSHER_FOLLOWER_TO_UPSTACK_TO_LOAD:
					load_to_upstack_to_load := FALSE;	 					
					
			END_CASE
		END_IF		
		
		IF	(active_cam <> next_cam)
			AND 
			connection_conditions
		THEN							
			connection_status_next := CSP_TRANSFER_CROSSPUSHER_STATUS_CONNECTION_CHANGE_CAM;
		END_IF
			
		IF	NOT connection_motorization_moving
		THEN
			connection_status_next := CSP_TRANSFER_CROSSPUSHER_STATUS_CONNECTION_DONE;
		END_IF
	
		
	CSP_TRANSFER_CROSSPUSHER_STATUS_CONNECTION_CHANGE_CAM:	
		
		IF next_cam = TRANSFER_CROSSPUSHER_FOLLOWER_TO_UPSTACK_TO_LOAD
		THEN
			engage_mode := AXIS_CAM_ENGAGE_ABSOLUTE;
			slave_offset := slave_offset_input;
		ELSIF next_cam = DWELL_CAM
		THEN
			engage_mode := AXIS_CAM_ENGAGE_RELATIVE;
			slave_offset := 0;
		END_IF
		
		IF NOT csp_transfer_crosspusher.reject_running
		THEN	
			axis_engage_cam(
				cam_id							:=	next_cam,	
				master_engage_mode				:=	AXIS_CAM_ENGAGE_ABSOLUTE,
				slave_engage_mode				:=	engage_mode,
				activation_mode					:=	AXIS_CAM_ACTIVATION_NEXT_CYCLE,
				activation_position				:=	0,
				master_scaling_mode				:=	AXIS_CAM_SCALING_MODE_USER_DEFINED,
				slave_scaling_mode				:=	AXIS_CAM_SCALING_MODE_USER_DEFINED,
				master_offset					:=	master_offset, 
				slave_offset					:=	slave_offset,
				master_scaling					:=	master_scaling,
				slave_scaling					:=	slave_scaling,
				interpolation_type				:=	AXIS_CAM_INTERPOLATION_SPLINE,	 
				master							:=	csp_transfer_crosspusher_virtualMaster.axis,
				CONVERSION_this					:=	axis);	
		END_IF
	
		IF	motorization_manager_is_starting(csp_main_motorization_manager.motm)
		THEN
			connection_status_next := CSP_TRANSFER_CROSSPUSHER_STATUS_CONNECTION_DONE;
		ELSE
			IF axis_is_cam_engaged(axis)
			THEN
				connection_status_next := CSP_TRANSFER_CROSSPUSHER_STATUS_CONNECTION_WAIT_NEW_CAM;
			END_IF
		END_IF
		
		
	CSP_TRANSFER_CROSSPUSHER_STATUS_CONNECTION_IMMEDIATE_CHANGE:
	
		axis_engage_cam(
			cam_id							:=	DWELL_CAM,	
			master_engage_mode				:=	AXIS_CAM_ENGAGE_ABSOLUTE,
			slave_engage_mode				:=	AXIS_CAM_ENGAGE_RELATIVE,
			activation_mode					:=	AXIS_CAM_ACTIVATION_IMMEDIATELY,
			activation_position				:=	0,
			master_scaling_mode				:=	AXIS_CAM_SCALING_MODE_USER_DEFINED,
			slave_scaling_mode				:=	AXIS_CAM_SCALING_MODE_USER_DEFINED,
			master_offset					:=	csp_transfer_crosspusher_virtualMaster.axis.actual_position,  
			slave_offset					:=	slave_offset,
			master_scaling					:=	master_scaling,
			slave_scaling					:=	slave_scale_test, //slave_scaling,
			interpolation_type				:=	AXIS_CAM_INTERPOLATION_SPLINE,	 
			master							:=	csp_transfer_crosspusher_virtualMaster.axis,
			CONVERSION_this					:=	axis);	
			
		next_cam := DWELL_CAM;
		active_cam := DWELL_CAM;			
			
		IF	motorization_manager_is_starting(csp_main_motorization_manager.motm)
		THEN
			connection_status_next := CSP_TRANSFER_CROSSPUSHER_STATUS_CONNECTION_DONE;
		ELSE
			IF csp_transfer_crosspusher.loader_clear
			THEN
				connection_status_next := CSP_TRANSFER_CROSSPUSHER_STATUS_CONNECTION_WAIT_NEW_CAM;
			END_IF
		END_IF	
		
		
	CSP_TRANSFER_CROSSPUSHER_STATUS_CONNECTION_WAIT_NEW_CAM:
	
		IF	active_cam = next_cam
		THEN
			CASE next_cam OF
				DWELL_CAM:
					activation_position := next_activation_position;
				
				FORWARD_CAM:
					activation_position := 0;					
			END_CASE
			connection_status_next := CSP_TRANSFER_CROSSPUSHER_STATUS_CONNECTION_CHECK_CHANGE_CAM;
		END_IF
		
		IF	NOT connection_motorization_moving
		THEN
			connection_status_next := CSP_TRANSFER_CROSSPUSHER_STATUS_CONNECTION_DONE;
		END_IF
		
		
	(* WAITS FOR REJECT SEQUENCE TO FINISH IF EVER GOES TO REJECT *)
	CSP_TRANSFER_CROSSPUSHER_STATUS_CONNECTION_WAIT_REJECT:
	
		IF axis_is_standstill(axis)
			AND csp_transfer_crosspusher.reject_done
		THEN
			active_cam := DWELL_CAM;
			next_cam := DWELL_CAM;
			connection_status_next := CSP_TRANSFER_CROSSPUSHER_STATUS_CONNECTION_ENGAGE;
		END_IF
		
				
	CSP_TRANSFER_CROSSPUSHER_STATUS_CONNECTION_DONE:    (* Connection done *)     
  
        connection_running := FALSE;
        connection_done := TRUE;
       
        motorization_conditioner_start_done(connection_done_motcond);
		IF	csp.o_machine_is_running//motorization_manager_is_execute(csp_main_motorization_manager.motm)
		THEN                       
			IF    active_cam <> next_cam
			THEN
				connection_status_next := CSP_TRANSFER_CROSSPUSHER_STATUS_CONNECTION_WAIT_NEW_CAM;
			ELSE
				connection_status_next := CSP_TRANSFER_CROSSPUSHER_STATUS_CONNECTION_CHECK_CHANGE_CAM;
			END_IF
        END_IF
       
	
	CSP_TRANSFER_CROSSPUSHER_STATUS_CONNECTION_ERROR:	(* Connection error *)	
	
		IF 	connection_running
			OR NOT axis_is_ok(FALSE, axis)
		THEN
			axis_disable(axis);
			connection_error := TRUE;						
		END_IF
		connection_running	:= FALSE;
		connection_done 	:= FALSE;	
		
		IF	connection_conditions
		THEN		
			connection_status_next := CSP_TRANSFER_CROSSPUSHER_STATUS_CONNECTION_START;
		END_IF
		
END_CASE

IF 	NOT debug_connection_state_machine
	OR
	debug_connection_machine_one_step	
THEN
	connection_status := connection_status_next;
	debug_connection_machine_one_step := FALSE;
END_IF

connection_motorization_moving	:= 
	motorization_manager_is_starting(csp_main_motorization_manager.motm)
	OR
	motorization_manager_is_execute(csp_main_motorization_manager.motm)
	OR
	motorization_manager_is_stopping(csp_main_motorization_manager.motm)
	OR
	motorization_manager_is_suspended(csp_main_motorization_manager.motm)
	OR
	motorization_manager_is_suspending(csp_main_motorization_manager.motm)
	OR
	motorization_manager_is_unsuspending(csp_main_motorization_manager.motm)
	OR 
	motorization_manager_is_holding(csp_main_motorization_manager.motm)
	OR
	motorization_manager_is_held(csp_main_motorization_manager.motm)
	OR
	motorization_manager_is_unholding(csp_main_motorization_manager.motm);
	
(* Connection timeout *)
IF	(connection_running
	AND NOT debug_connection_state_machine)	
	OR connection_error
	AND NOT csp_transfer_crosspusher.reject_running 
THEN
	IF	timer_is_expired(connection_time_out_tmr)
	THEN
		process_message_set(1, connection_status, 0, connection_faulted_aem);
	END_IF
ELSE
	timer_restart(10000, connection_time_out_tmr);
END_IF
END_ACTION

ACTION phase:
phase_conditions :=
	axis_is_ok(FALSE, axis)
	AND
	process_is_ready(prc)
	AND
	process_subtree_is_ready(prc)
	AND
	servo_on_condition
	AND				
	NOT csp_transfer_main_brand.cam_data_changed
	AND
	NOT disable_req
	AND						
	NOT jog_manager_is_jog_axis_active(SMTR41503_TRANSFER_CROSSPUSHER_FOLLOWER, csp_main_jogManager.jog_manager_real);				
	
(* phase_done reset *)
IF	phase_done
	AND
	NOT phase_conditions
	AND 
	NOT csp.o_machine_is_running
THEN
	axis_disable(axis);
	phase_done:= FALSE;
END_IF

(* Exit condition *)
IF 	NOT phase_conditions
THEN
	phase_status_next := CSP_TRANSFER_CROSSPUSHER_PHASE_STATUS_ERROR;
	phase_status := phase_status_next;	
END_IF

(*************** MACHINE STATUS ***************)
CASE phase_status OF

	CSP_TRANSFER_CROSSPUSHER_PHASE_STATUS_START:	(* Start phasing *)
	
		IF motorization_manager_is_starting(csp_main_motorization_manager.motm) 
			AND csp_transfer_crosspusher_virtualMaster.phase_done
			AND csp_transfer_crosspusher_virtualMaster.connection_done
			AND NOT csp_transfer_crosspusher.reject_running
		THEN
			phase_running := TRUE;			
			phase_status_next := CSP_TRANSFER_CROSSPUSHER_PHASE_STATUS_DISABLE;
		END_IF
		
				
	CSP_TRANSFER_CROSSPUSHER_PHASE_STATUS_DISABLE:
	
		axis_disable(axis);		
		IF 	axis_is_disabled(axis)
		THEN
			phase_status_next := CSP_TRANSFER_CROSSPUSHER_PHASE_STATUS_ENABLE;
		END_IF
		
		
	CSP_TRANSFER_CROSSPUSHER_PHASE_STATUS_ENABLE:
	
		axis_enable(axis);		
		IF 	axis_is_enabled(axis)
		THEN
			phase_status_next := CSP_TRANSFER_CROSSPUSHER_PHASE_STATUS_ENABLED;
		END_IF
		
		
	CSP_TRANSFER_CROSSPUSHER_PHASE_STATUS_ENABLED:
	
		IF 	axis_is_standstill(axis) 
		THEN
			phase_status_next := CSP_TRANSFER_CROSSPUSHER_PHASE_STATUS_CALCULATE_SLAVE_POSITION_REQUEST;								
		END_IF
		
		
	CSP_TRANSFER_CROSSPUSHER_PHASE_STATUS_CALCULATE_SLAVE_POSITION_REQUEST:
	
		slave_position_has_been_calculated := FALSE;
		(* CHECK THE LOADER TO SEE IF IT IS DONE OR IS IN THE WAY AND CHANGE CAM *)
		IF csp_case_loader_pusher.fsm_status > CSP_CASE_LOADER_STATUS_PHASED
		THEN		
			(* Gets the position of the master axis *)
			axis_calculate_cam_slave_master_position_deg := 
				LMOD(axis_get_actual_modulo_position(csp_transfer_crosspusher_virtualMaster.axis)
				+ home_position_master_offset_deg, G_MODULO_360_DEG);
				
			(* Gets cam data for slave axis to master *)
			IF axis_calculate_cam_slave_dynamics_data(
				cam_id := active_cam,
				master_scaling := master_scaling,
				master_position := axis_calculate_cam_slave_master_position_deg,
				slave_scaling := slave_scaling,
				CONVERSION_this := axis)
			THEN
				timer_restart(phase_delay, phase_delay_tmr);
				phase_status_next := CSP_TRANSFER_CROSSPUSHER_PHASE_STATUS_CALCULATING_SLAVE_POSITION;
			END_IF
		END_IF
				
	
	CSP_TRANSFER_CROSSPUSHER_PHASE_STATUS_CALCULATING_SLAVE_POSITION:
	
		IF 	axis_cam_slave_dynamics_data_calculated(axis)
			AND timer_is_expired(phase_delay_tmr)
		THEN
			IF active_cam = DWELL_CAM
			THEN
				axis_calculated_cam_slave_position_deg := axis_get_cam_slave_dynamics_position(axis) + slave_scaling + slave_offset; //slave_scaling; (* RMH - Unsure if this is the safest approach to phasing followering to load position at startup *)
			ELSE
				axis_calculated_cam_slave_position_deg := axis_get_cam_slave_dynamics_position(axis);
			END_IF
			
			slave_position_has_been_calculated := TRUE;
			
			IF axis.actual_position > axis_calculated_cam_slave_position_deg
			THEN 
				direction_FWD := FALSE;	// backward
			ELSIF axis.actual_position < axis_calculated_cam_slave_position_deg
			THEN
				direction_FWD := TRUE; //forward
			END_IF
			
			phase_status_next := CSP_TRANSFER_PHASE_STATUS_REQUEST;				
		END_IF
		
		
	CSP_TRANSFER_PHASE_STATUS_REQUEST:
		
